Yaskawa INFORM job: aprem3TRJ4.JBI

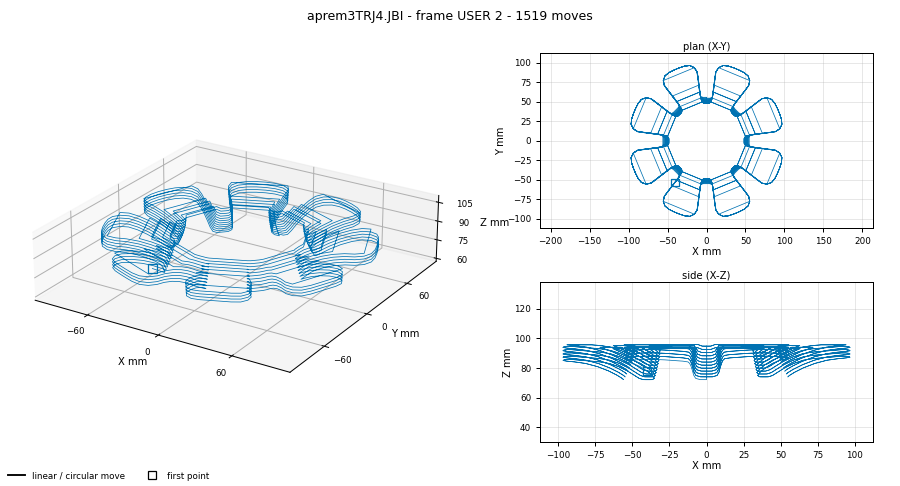
[picture p0: tool path of aprem3TRJ4.JBI in frame USER 2, 1519 of 1519 moves have a stored position in this frame; points joined in program order, loops and branches not executed]
/JOB
//NAME aprem3TRJ4
///FOLDERNAME DEMO
//POS
///NPOS 1519,0,1519,0,0,0
///USER 2
///TOOL 7
///POSTYPE USER
///RECTAN
///RCONF 1,0,0,0,0,0,0,0,0,0,0,0,0,0,0,0,0,0,0,0,0,0,0,0
C00000=-40.007,-53.324,78.036,177.7295,-3.1005,-14256.8795
C00001=-36.517,-48.718,75.143,178.8242,-1.7083,-14256.8537
C00002=-35.037,-45.351,73.015,-179.8825,17.3486,-14257.6887
C00003=-36.538,-42.505,72.166,160.0580,24.5520,-14260.6829
C00004=-38.303,-40.803,72.129,156.0408,22.3844,-14263.1899
C00005=-39.567,-39.567,72.154,156.8171,23.1818,-14265.0000
C00006=-40.803,-38.303,72.129,157.6162,23.9597,-14266.8101
C00007=-42.506,-36.538,72.166,155.4471,19.9396,-14269.3178
C00008=-45.352,-35.037,73.015,162.6519,-0.1179,-14272.3119
C00009=-48.718,-36.517,75.143,-178.2917,1.1758,-14273.1463
C00010=-53.324,-40.007,78.036,-176.8995,2.2705,-14273.1205
C00011=-59.196,-44.618,80.927,-176.4745,2.6327,-14272.9934
C00012=-65.578,-49.604,83.062,-176.2466,2.8111,-14272.8957
C00013=-71.524,-53.949,84.088,-176.0077,2.0393,-14272.9735
C00014=-77.795,-55.184,84.621,-177.1914,-0.2563,-14274.6500
C00015=-83.601,-53.037,85.050,-178.9039,-0.7847,-14277.6087
C00016=-87.741,-47.957,85.481,-179.9577,-0.0772,-14281.3401
C00017=-90.934,-41.602,85.762,-179.9958,-0.0092,-14285.4161
C00018=-93.717,-34.883,85.762,-179.9965,-0.0095,-14289.5839
C00019=-95.953,-28.131,85.481,-179.9754,-0.0845,-14293.6602
C00020=-96.617,-21.612,85.050,179.7797,-1.3299,-14297.3912
C00021=-94.030,-15.989,84.621,178.1943,-2.1678,-14300.3496
C00022=-88.723,-12.427,84.088,175.7377,-1.3847,-14302.0267
C00023=-81.446,-11.295,83.062,175.3629,-0.6685,-14302.1045
C00024=-73.408,-10.308,80.927,175.6494,-0.6331,-14302.0068
C00025=-65.995,-9.417,78.036,176.2047,-0.5882,-14301.8791
C00026=-60.270,-8.627,75.143,177.9610,-0.3768,-14301.8541
C00027=-56.844,-7.293,73.015,-167.4643,12.3773,-14302.6890
C00028=-55.892,-4.219,72.166,-176.1973,30.0956,-14305.6832
C00029=-55.936,-1.768,72.129,178.6826,31.1925,-14308.1896
C00030=-55.957,0.000,72.154,179.9991,31.1998,-14310.0000
C00031=-55.936,1.767,72.129,-178.6816,31.1926,-14311.8094
C00032=-55.892,4.220,72.166,176.1946,30.0948,-14314.3178
C00033=-56.844,7.293,73.015,167.4645,12.3766,-14317.3110
C00034=-60.270,8.627,75.143,-177.9610,-0.3768,-14318.1459
C00035=-65.995,9.417,78.036,-176.2047,-0.5882,-14318.1209
C00036=-73.408,10.308,80.927,-175.6494,-0.6331,-14317.9932
C00037=-81.446,11.295,83.062,-175.3629,-0.6685,-14317.8955
C00038=-88.723,12.427,84.088,-175.7377,-1.3847,-14317.9733
C00039=-94.030,15.989,84.621,-178.1943,-2.1678,-14319.6504
C00040=-96.617,21.612,85.050,-179.7797,-1.3299,-14322.6088
C00041=-95.953,28.131,85.481,179.9754,-0.0845,-14326.3398
C00042=-93.717,34.883,85.762,179.9965,-0.0095,-14330.4161
C00043=-90.934,41.602,85.762,179.9958,-0.0092,-14334.5839
C00044=-87.741,47.957,85.481,179.9577,-0.0772,-14338.6599
C00045=-83.601,53.037,85.050,178.9039,-0.7847,-14342.3913
C00046=-77.795,55.184,84.621,177.1914,-0.2563,-14345.3500
C00047=-71.524,53.949,84.088,176.0077,2.0393,-14347.0265
C00048=-65.578,49.604,83.062,176.2466,2.8111,-14347.1043
C00049=-59.196,44.618,80.927,176.4745,2.6327,-14347.0066
C00050=-53.324,40.007,78.036,176.8995,2.2705,-14346.8795
C00051=-48.718,36.517,75.143,178.2917,1.1758,-14346.8537
C00052=-45.351,35.037,73.015,-162.6514,-0.1175,-14347.6887
C00053=-42.505,36.538,72.166,-155.4480,19.9420,-14350.6829
C00054=-40.803,38.303,72.129,-157.6156,23.9592,-14353.1899
C00055=-39.567,39.567,72.154,-156.8182,23.1829,-14355.0000
C00056=-38.303,40.803,72.129,-156.0403,22.3838,-14356.8101
C00057=-36.538,42.506,72.166,-160.0604,24.5529,-14359.3178
C00058=-35.037,45.352,73.015,179.8821,17.3481,-14362.3119
C00059=-36.517,48.718,75.143,-178.8242,-1.7083,-14363.1463
C00060=-40.007,53.324,78.036,-177.7295,-3.1005,-14363.1205
C00061=-44.618,59.196,80.927,-177.3673,-3.5255,-14362.9934
C00062=-49.604,65.578,83.062,-177.1889,-3.7534,-14362.8957
C00063=-53.949,71.524,84.088,-177.9607,-3.9923,-14362.9735
C00064=-55.184,77.795,84.621,179.7437,-2.8086,-14364.6500
C00065=-53.037,83.601,85.050,179.2153,-1.0961,-14367.6087
C00066=-47.957,87.741,85.481,179.9228,-0.0423,-14371.3401
C00067=-41.602,90.934,85.762,179.9908,-0.0042,-14375.4161
C00068=-34.883,93.717,85.762,179.9905,-0.0035,-14379.5839
C00069=-28.131,95.953,85.481,179.9155,-0.0246,-14383.6602
C00070=-21.612,96.617,85.050,178.6701,0.2203,-14387.3912
C00071=-15.989,94.030,84.621,177.8322,1.8057,-14390.3496
C00072=-12.427,88.723,84.088,178.6153,4.2623,-14392.0267
C00073=-11.295,81.446,83.062,179.3315,4.6371,-14392.1045
C00074=-10.308,73.408,80.927,179.3669,4.3506,-14392.0068
C00075=-9.417,65.995,78.036,179.4118,3.7953,-14391.8791
C00076=-8.627,60.270,75.143,179.6232,2.0390,-14391.8541
C00077=-7.293,56.844,73.015,-167.6234,-12.5355,-14392.6890
C00078=-4.220,55.892,72.166,-149.9052,-3.8054,-14395.6822
C00079=-1.767,55.936,72.129,-148.8074,1.3184,-14398.1906
C00080=0.000,55.957,72.154,-148.8002,-0.0009,-14400.0000
C00081=0.000,54.840,74.049,-150.2606,-0.0009,-14400.0000
C00082=1.666,54.823,74.024,-150.2652,-1.1897,-14401.7406
C00083=4.048,54.790,74.062,-151.4249,3.8705,-14404.2255
C00084=7.088,55.804,74.943,-168.9167,11.6638,-14407.2387
C00085=8.393,59.388,77.145,179.6271,-2.1340,-14408.0440
C00086=9.180,65.335,80.122,179.4707,-3.5331,-14407.9981
C00087=10.089,72.980,83.074,179.4510,-3.8704,-14407.8709
C00088=11.094,81.206,85.240,179.4410,-3.9838,-14407.7793
C00089=12.226,88.613,86.276,178.8532,-3.5972,-14407.8555
C00090=15.808,94.009,86.813,178.1980,-1.5172,-14409.5452
C00091=21.475,96.642,87.246,178.9013,-0.1852,-14412.5282
C00092=28.048,95.980,87.679,179.9308,0.0202,-14416.2898
C00093=34.856,93.728,87.962,179.9923,0.0029,-14420.3994
C00094=41.629,90.922,87.962,179.9925,0.0034,-14424.6009
C00095=48.035,87.701,87.679,179.9368,0.0347,-14428.7101
C00096=53.151,83.521,87.246,179.3540,0.9079,-14432.4718
C00097=55.296,77.652,86.813,179.7985,2.3464,-14435.4547
C00098=54.014,71.304,86.276,-178.2646,3.3541,-14437.1446
C00099=49.577,65.266,85.240,-177.5752,3.2135,-14437.2208
C00100=44.470,58.738,83.074,-177.6486,3.1261,-14437.1290
C00101=39.708,52.690,80.122,-177.8738,2.8733,-14437.0022
C00102=36.059,47.928,77.145,-178.7542,1.7728,-14436.9563
C00103=34.447,44.472,74.943,179.5730,-15.8802,-14437.7605
C00104=35.880,41.605,74.062,-161.3614,-23.4111,-14440.7744
C00105=37.588,39.944,74.024,-157.2868,-21.2665,-14443.2595
C00106=38.778,38.778,74.049,-158.0022,-21.9968,-14445.0000
C00107=39.943,37.588,74.024,-158.7340,-22.7138,-14446.7398
C00108=41.605,35.880,74.062,-156.5881,-18.6363,-14449.2256
C00109=44.472,34.447,74.943,-164.1205,0.4274,-14452.2395
C00110=47.928,36.059,77.145,178.2272,-1.2458,-14453.0437
C00111=52.690,39.708,80.122,177.1267,-2.1262,-14452.9978
C00112=58.738,44.470,83.074,176.8739,-2.3514,-14452.8710
C00113=65.266,49.577,85.240,176.7865,-2.4248,-14452.7792
C00114=71.304,54.014,86.276,176.6459,-1.7354,-14452.8554
C00115=77.652,55.296,86.813,177.6536,0.2015,-14454.5453
C00116=83.521,53.151,87.246,179.0921,0.6460,-14457.5282
C00117=87.701,48.035,87.679,179.9653,0.0632,-14461.2899
C00118=90.922,41.629,87.962,179.9966,0.0075,-14465.3991
C00119=93.728,34.856,87.962,179.9971,0.0077,-14469.6006
C00120=95.980,28.048,87.679,179.9798,0.0692,-14473.7102
C00121=96.642,21.475,87.246,-179.8148,1.0987,-14477.4718
C00122=94.009,15.808,86.813,-178.4828,1.8020,-14480.4548
C00123=88.613,12.226,86.276,-176.4028,1.1468,-14482.1445
C00124=81.206,11.094,85.240,-176.0162,0.5590,-14482.2207
C00125=72.980,10.089,83.074,-176.1296,0.5490,-14482.1291
C00126=65.335,9.180,80.122,-176.4669,0.5293,-14482.0019
C00127=59.388,8.393,77.145,-177.8660,0.3729,-14481.9560
C00128=55.804,7.088,74.943,168.3362,-11.0833,-14482.7613
C00129=54.790,4.048,74.062,176.1295,-28.5751,-14485.7745
C00130=54.823,1.666,74.024,-178.8103,-29.7348,-14488.2594
C00131=54.840,0.000,74.049,-179.9991,-29.7394,-14490.0000
C00132=54.823,-1.665,74.024,178.8094,-29.7348,-14491.7396
C00133=54.790,-4.048,74.062,-176.1270,-28.5741,-14494.2255
C00134=55.804,-7.088,74.943,-168.3364,-11.0826,-14497.2387
C00135=59.388,-8.393,77.145,177.8660,0.3729,-14498.0440
C00136=65.335,-9.180,80.122,176.4669,0.5293,-14497.9981
C00137=72.980,-10.089,83.074,176.1296,0.5490,-14497.8709
C00138=81.206,-11.094,85.240,176.0162,0.5590,-14497.7793
C00139=88.613,-12.226,86.276,176.4028,1.1468,-14497.8555
C00140=94.009,-15.808,86.813,178.4828,1.8020,-14499.5452
C00141=96.642,-21.475,87.246,179.8148,1.0987,-14502.5282
C00142=95.980,-28.048,87.679,-179.9798,0.0692,-14506.2898
C00143=93.728,-34.856,87.962,-179.9971,0.0077,-14510.3994
C00144=90.922,-41.629,87.962,-179.9966,0.0075,-14514.6009
C00145=87.701,-48.035,87.679,-179.9653,0.0632,-14518.7101
C00146=83.521,-53.151,87.246,-179.0921,0.6460,-14522.4718
C00147=77.652,-55.296,86.813,-177.6536,0.2015,-14525.4547
C00148=71.304,-54.014,86.276,-176.6459,-1.7354,-14527.1446
C00149=65.266,-49.577,85.240,-176.7865,-2.4248,-14527.2208
C00150=58.738,-44.470,83.074,-176.8739,-2.3514,-14527.1290
C00151=52.690,-39.708,80.122,-177.1267,-2.1262,-14527.0022
C00152=47.928,-36.059,77.145,-178.2272,-1.2458,-14526.9563
C00153=44.472,-34.447,74.943,164.1198,0.4270,-14527.7605
C00154=41.605,-35.880,74.062,156.5889,-18.6386,-14530.7744
C00155=39.944,-37.588,74.024,158.7335,-22.7132,-14533.2595
C00156=38.778,-38.778,74.049,158.0032,-21.9978,-14535.0000
C00157=37.588,-39.943,74.024,157.2862,-21.2660,-14536.7398
C00158=35.880,-41.605,74.062,161.3637,-23.4119,-14539.2256
C00159=34.447,-44.472,74.943,-179.5726,-15.8795,-14542.2395
C00160=36.059,-47.928,77.145,178.7542,1.7728,-14543.0437
C00161=39.708,-52.690,80.122,177.8738,2.8733,-14542.9978
C00162=44.470,-58.738,83.074,177.6486,3.1261,-14542.8710
C00163=49.577,-65.266,85.240,177.5752,3.2135,-14542.7792
C00164=54.014,-71.304,86.276,178.2646,3.3541,-14542.8554
C00165=55.296,-77.652,86.813,-179.7985,2.3464,-14544.5453
C00166=53.151,-83.521,87.246,-179.3540,0.9079,-14547.5282
C00167=48.035,-87.701,87.679,-179.9368,0.0347,-14551.2899
C00168=41.629,-90.922,87.962,-179.9925,0.0034,-14555.3991
C00169=34.856,-93.728,87.962,-179.9923,0.0029,-14559.6006
C00170=28.048,-95.980,87.679,-179.9308,0.0202,-14563.7102
C00171=21.475,-96.642,87.246,-178.9013,-0.1852,-14567.4718
C00172=15.808,-94.009,86.813,-178.1980,-1.5172,-14570.4548
C00173=12.226,-88.613,86.276,-178.8532,-3.5972,-14572.1445
C00174=11.094,-81.206,85.240,-179.4410,-3.9838,-14572.2207
C00175=10.089,-72.980,83.074,-179.4510,-3.8704,-14572.1291
C00176=9.180,-65.335,80.122,-179.4707,-3.5331,-14572.0019
C00177=8.393,-59.388,77.145,-179.6271,-2.1340,-14571.9560
C00178=7.088,-55.804,74.943,168.9167,11.6638,-14572.7613
C00179=4.048,-54.790,74.062,151.4249,3.8705,-14575.7745
C00180=1.666,-54.823,74.024,150.2652,-1.1897,-14578.2594
C00181=0.000,-54.840,74.049,150.2606,-0.0009,-14580.0000
C00182=0.000,-54.840,74.049,150.2606,-0.0009,-14580.0000
C00183=-1.665,-54.823,74.024,150.2652,1.1906,-14581.7396
C00184=-4.048,-54.790,74.062,151.4259,-3.8730,-14584.2255
C00185=-7.088,-55.804,74.943,168.9174,-11.6636,-14587.2387
C00186=-8.393,-59.388,77.145,-179.6271,2.1340,-14588.0440
C00187=-9.180,-65.335,80.122,-179.4707,3.5331,-14587.9981
C00188=-10.089,-72.980,83.074,-179.4510,3.8704,-14587.8709
C00189=-11.094,-81.206,85.240,-179.4410,3.9838,-14587.7793
C00190=-12.226,-88.613,86.276,-178.8532,3.5972,-14587.8555
C00191=-15.808,-94.009,86.813,-178.1980,1.5172,-14589.5452
C00192=-21.475,-96.642,87.246,-178.9013,0.1852,-14592.5282
C00193=-28.048,-95.980,87.679,-179.9308,-0.0202,-14596.2898
C00194=-34.856,-93.728,87.962,-179.9923,-0.0029,-14600.3994
C00195=-41.629,-90.922,87.962,-179.9925,-0.0034,-14604.6009
C00196=-48.035,-87.701,87.679,-179.9368,-0.0347,-14608.7101
C00197=-53.151,-83.521,87.246,-179.3540,-0.9079,-14612.4718
C00198=-55.296,-77.652,86.813,-179.7985,-2.3464,-14615.4547
C00199=-54.014,-71.304,86.276,178.2646,-3.3541,-14617.1446
C00200=-49.577,-65.266,85.240,177.5752,-3.2135,-14617.2208
C00201=-44.470,-58.738,83.074,177.6486,-3.1261,-14617.1290
C00202=-39.708,-52.690,80.122,177.8738,-2.8733,-14617.0022
C00203=-36.059,-47.928,77.145,178.7542,-1.7728,-14616.9563
C00204=-34.447,-44.472,74.943,-179.5730,15.8802,-14617.7605
C00205=-35.880,-41.605,74.062,161.3614,23.4111,-14620.7744
C00206=-37.588,-39.944,74.024,157.2868,21.2665,-14623.2595
C00207=-38.778,-38.778,74.049,158.0022,21.9968,-14625.0000
C00208=-39.943,-37.588,74.024,158.7340,22.7138,-14626.7398
C00209=-41.605,-35.880,74.062,156.5881,18.6363,-14629.2256
C00210=-44.472,-34.447,74.943,164.1205,-0.4274,-14632.2395
C00211=-47.928,-36.059,77.145,-178.2272,1.2458,-14633.0437
C00212=-52.690,-39.708,80.122,-177.1267,2.1262,-14632.9978
C00213=-58.738,-44.470,83.074,-176.8739,2.3514,-14632.8710
C00214=-65.266,-49.577,85.240,-176.7865,2.4248,-14632.7792
C00215=-71.304,-54.014,86.276,-176.6459,1.7354,-14632.8554
C00216=-77.652,-55.296,86.813,-177.6536,-0.2015,-14634.5453
C00217=-83.521,-53.151,87.246,-179.0921,-0.6460,-14637.5282
C00218=-87.701,-48.035,87.679,-179.9653,-0.0632,-14641.2899
C00219=-90.922,-41.629,87.962,-179.9966,-0.0075,-14645.3991
C00220=-93.728,-34.856,87.962,-179.9971,-0.0077,-14649.6006
C00221=-95.980,-28.048,87.679,-179.9798,-0.0692,-14653.7102
C00222=-96.642,-21.475,87.246,179.8148,-1.0987,-14657.4718
C00223=-94.009,-15.808,86.813,178.4828,-1.8020,-14660.4548
C00224=-88.613,-12.226,86.276,176.4028,-1.1468,-14662.1445
C00225=-81.206,-11.094,85.240,176.0162,-0.5590,-14662.2207
C00226=-72.980,-10.089,83.074,176.1296,-0.5490,-14662.1291
C00227=-65.335,-9.180,80.122,176.4669,-0.5293,-14662.0019
C00228=-59.388,-8.393,77.145,177.8660,-0.3729,-14661.9560
C00229=-55.804,-7.088,74.943,-168.3362,11.0833,-14662.7613
C00230=-54.790,-4.048,74.062,-176.1295,28.5751,-14665.7745
C00231=-54.823,-1.666,74.024,178.8103,29.7348,-14668.2594
C00232=-54.840,0.000,74.049,179.9991,29.7394,-14670.0000
C00233=-54.823,1.665,74.024,-178.8094,29.7348,-14671.7396
C00234=-54.790,4.048,74.062,176.1270,28.5741,-14674.2255
C00235=-55.804,7.088,74.943,168.3364,11.0826,-14677.2387
C00236=-59.388,8.393,77.145,-177.8660,-0.3729,-14678.0440
C00237=-65.335,9.180,80.122,-176.4669,-0.5293,-14677.9981
C00238=-72.980,10.089,83.074,-176.1296,-0.5490,-14677.8709
C00239=-81.206,11.094,85.240,-176.0162,-0.5590,-14677.7793
C00240=-88.613,12.226,86.276,-176.4028,-1.1468,-14677.8555
C00241=-94.009,15.808,86.813,-178.4828,-1.8020,-14679.5452
C00242=-96.642,21.475,87.246,-179.8148,-1.0987,-14682.5282
C00243=-95.980,28.048,87.679,179.9798,-0.0692,-14686.2898
C00244=-93.728,34.856,87.962,179.9971,-0.0077,-14690.3994
C00245=-90.922,41.629,87.962,179.9966,-0.0075,-14694.6009
C00246=-87.701,48.035,87.679,179.9653,-0.0632,-14698.7101
C00247=-83.521,53.151,87.246,179.0921,-0.6460,-14702.4718
C00248=-77.652,55.296,86.813,177.6536,-0.2015,-14705.4547
C00249=-71.304,54.014,86.276,176.6459,1.7354,-14707.1446
C00250=-65.266,49.577,85.240,176.7865,2.4248,-14707.2208
C00251=-58.738,44.470,83.074,176.8739,2.3514,-14707.1290
C00252=-52.690,39.708,80.122,177.1267,2.1262,-14707.0022
C00253=-47.928,36.059,77.145,178.2272,1.2458,-14706.9563
C00254=-44.472,34.447,74.943,-164.1198,-0.4270,-14707.7605
C00255=-41.605,35.880,74.062,-156.5889,18.6386,-14710.7744
C00256=-39.944,37.588,74.024,-158.7335,22.7132,-14713.2595
C00257=-38.778,38.778,74.049,-158.0032,21.9978,-14715.0000
C00258=-37.588,39.943,74.024,-157.2862,21.2660,-14716.7398
C00259=-35.880,41.605,74.062,-161.3637,23.4119,-14719.2256
C00260=-34.447,44.472,74.943,179.5726,15.8795,-14722.2395
C00261=-36.059,47.928,77.145,-178.7542,-1.7728,-14723.0437
C00262=-39.708,52.690,80.122,-177.8738,-2.8733,-14722.9978
C00263=-44.470,58.738,83.074,-177.6486,-3.1261,-14722.8710
C00264=-49.577,65.266,85.240,-177.5752,-3.2135,-14722.7792
C00265=-54.014,71.304,86.276,-178.2646,-3.3541,-14722.8554
C00266=-55.296,77.652,86.813,179.7985,-2.3464,-14724.5453
C00267=-53.151,83.521,87.246,179.3540,-0.9079,-14727.5282
C00268=-48.035,87.701,87.679,179.9368,-0.0347,-14731.2899
C00269=-41.629,90.922,87.962,179.9925,-0.0034,-14735.3991
C00270=-34.856,93.728,87.962,179.9923,-0.0029,-14739.6006
C00271=-28.048,95.980,87.679,179.9308,-0.0202,-14743.7102
C00272=-21.475,96.642,87.246,178.9013,0.1852,-14747.4718
C00273=-15.808,94.009,86.813,178.1980,1.5172,-14750.4548
C00274=-12.226,88.613,86.276,178.8532,3.5972,-14752.1445
C00275=-11.094,81.206,85.240,179.4410,3.9838,-14752.2207
C00276=-10.089,72.980,83.074,179.4510,3.8704,-14752.1291
C00277=-9.180,65.335,80.122,179.4707,3.5331,-14752.0019
C00278=-8.393,59.388,77.145,179.6271,2.1340,-14751.9560
C00279=-7.088,55.804,74.943,-168.9174,-11.6636,-14752.7613
C00280=-4.048,54.790,74.062,-151.4259,-3.8730,-14755.7745
C00281=-1.665,54.823,74.024,-150.2652,1.1906,-14758.2604
C00282=0.000,54.840,74.049,-150.2606,-0.0009,-14760.0000
C00283=0.000,53.776,75.975,-151.9017,-0.0008,-14760.0000
C00284=1.568,53.762,75.948,-151.9034,-1.0593,-14761.6706
C00285=3.884,53.739,75.988,-153.1148,3.8750,-14764.1339
C00286=6.894,54.818,76.900,-170.1649,10.7294,-14767.1680
C00287=8.175,58.565,79.173,179.6434,-2.1517,-14767.9465
C00288=8.965,64.737,82.228,179.5331,-3.2135,-14767.8844
C00289=9.898,72.606,85.234,179.5371,-3.3364,-14767.7630
C00290=10.924,81.005,87.424,179.5509,-3.2738,-14767.6803
C00291=12.061,88.524,88.468,179.0976,-2.8742,-14767.7585
C00292=15.662,93.991,89.008,178.5900,-1.1973,-14769.4604
C00293=21.365,96.662,89.443,179.1515,-0.1450,-14772.4636
C00294=27.983,96.002,89.878,179.9474,0.0153,-14776.2505
C00295=34.834,93.736,90.162,179.9942,0.0022,-14780.3860
C00296=41.650,90.913,90.162,179.9944,0.0026,-14784.6140
C00297=48.097,87.670,89.878,179.9520,0.0264,-14788.7498
C00298=53.243,83.458,89.443,179.5025,0.7025,-14792.5363
C00299=55.387,77.537,89.008,179.8495,1.8433,-14795.5394
C00300=54.067,71.124,88.468,-178.6043,2.6703,-14797.2413
C00301=49.554,65.004,87.424,-178.0010,2.6331,-14797.3191
C00302=44.341,58.339,85.234,-177.9664,2.6872,-14797.2369
C00303=39.437,52.115,82.228,-178.0562,2.6030,-14797.1159
C00304=35.631,47.192,79.173,-178.7302,1.7738,-14797.0536
C00305=33.888,43.637,76.900,179.3468,-14.3899,-14797.8325
C00306=35.253,40.746,75.988,-162.7447,-22.1169,-14800.8660
C00307=36.906,39.124,75.948,-158.6653,-20.0234,-14803.3290
C00308=38.025,38.025,75.975,-159.3164,-20.6826,-14805.0000
C00309=39.124,36.906,75.948,-159.9771,-21.3352,-14806.6710
C00310=40.746,35.253,75.988,-157.8823,-17.2529,-14809.1340
C00311=43.637,33.888,76.901,-165.6107,0.6536,-14812.1675
C00312=47.192,35.631,79.173,178.2262,-1.2698,-14812.9464
C00313=52.115,39.437,82.228,177.3970,-1.9438,-14812.8841
C00314=58.339,44.341,85.234,177.3128,-2.0336,-14812.7631
C00315=65.004,49.554,87.424,177.3669,-1.9990,-14812.6809
C00316=71.124,54.067,88.468,177.3297,-1.3957,-14812.7587
C00317=77.537,55.387,89.008,178.1567,0.1505,-14814.4606
C00318=83.458,53.243,89.443,179.2975,0.4975,-14817.4637
C00319=87.670,48.097,89.878,179.9736,0.0480,-14821.2502
C00320=90.913,41.650,90.162,179.9974,0.0056,-14825.3860
C00321=93.736,34.834,90.162,179.9978,0.0058,-14829.6140
C00322=96.002,27.983,89.878,179.9847,0.0526,-14833.7495
C00323=96.662,21.365,89.443,-179.8550,0.8485,-14837.5364
C00324=93.991,15.662,89.008,-178.8027,1.4100,-14840.5396
C00325=88.524,12.061,88.468,-177.1258,0.9024,-14842.2415
C00326=81.005,10.924,87.424,-176.7262,0.4491,-14842.3197
C00327=72.606,9.898,85.234,-176.6636,0.4629,-14842.2370
C00328=64.737,8.965,82.228,-176.7865,0.4669,-14842.1156
C00329=58.565,8.175,79.173,-177.8483,0.3566,-14842.0535
C00330=54.818,6.894,76.900,169.2706,-9.8351,-14842.8320
C00331=53.739,3.884,75.988,176.1250,-26.8852,-14845.8661
C00332=53.762,1.568,75.948,-178.9407,-28.0966,-14848.3294
C00333=53.776,0.000,75.975,-179.9992,-28.0983,-14850.0000
C00334=53.762,-1.568,75.948,178.9399,-28.0967,-14851.6706
C00335=53.739,-3.885,75.988,-176.1225,-26.8842,-14854.1349
C00336=54.819,-6.894,76.901,-169.2709,-9.8343,-14857.1678
C00337=58.565,-8.175,79.173,177.8483,0.3566,-14857.9465
C00338=64.737,-8.965,82.228,176.7865,0.4669,-14857.8844
C00339=72.606,-9.898,85.234,176.6636,0.4629,-14857.7630
C00340=81.005,-10.924,87.424,176.7262,0.4491,-14857.6803
C00341=88.524,-12.061,88.468,177.1258,0.9024,-14857.7585
C00342=93.991,-15.662,89.008,178.8027,1.4100,-14859.4604
C00343=96.662,-21.365,89.443,179.8550,0.8485,-14862.4636
C00344=96.002,-27.983,89.878,-179.9847,0.0526,-14866.2505
C00345=93.736,-34.834,90.162,-179.9978,0.0058,-14870.3860
C00346=90.913,-41.650,90.162,-179.9974,0.0056,-14874.6140
C00347=87.670,-48.097,89.878,-179.9736,0.0480,-14878.7498
C00348=83.458,-53.243,89.443,-179.2975,0.4975,-14882.5363
C00349=77.537,-55.387,89.008,-178.1567,0.1505,-14885.5394
C00350=71.124,-54.067,88.468,-177.3297,-1.3957,-14887.2413
C00351=65.004,-49.554,87.424,-177.3669,-1.9990,-14887.3191
C00352=58.339,-44.341,85.234,-177.3128,-2.0336,-14887.2369
C00353=52.115,-39.437,82.228,-177.3970,-1.9438,-14887.1159
C00354=47.192,-35.631,79.173,-178.2262,-1.2698,-14887.0536
C00355=43.637,-33.888,76.900,165.6101,0.6532,-14887.8325
C00356=40.746,-35.253,75.988,157.8831,-17.2553,-14890.8660
C00357=39.124,-36.906,75.948,159.9766,-21.3347,-14893.3290
C00358=38.025,-38.025,75.975,159.3174,-20.6836,-14895.0000
C00359=36.906,-39.124,75.948,158.6648,-20.0229,-14896.6710
C00360=35.253,-40.746,75.988,162.7471,-22.1177,-14899.1340
C00361=33.888,-43.637,76.901,-179.3464,-14.3893,-14902.1675
C00362=35.631,-47.192,79.173,178.7302,1.7738,-14902.9464
C00363=39.437,-52.115,82.228,178.0562,2.6030,-14902.8841
C00364=44.341,-58.339,85.234,177.9664,2.6872,-14902.7631
C00365=49.554,-65.004,87.424,178.0010,2.6331,-14902.6809
C00366=54.067,-71.124,88.468,178.6043,2.6703,-14902.7587
C00367=55.387,-77.537,89.008,-179.8495,1.8433,-14904.4606
C00368=53.243,-83.458,89.443,-179.5025,0.7025,-14907.4637
C00369=48.097,-87.670,89.878,-179.9520,0.0264,-14911.2502
C00370=41.650,-90.913,90.162,-179.9944,0.0026,-14915.3860
C00371=34.834,-93.736,90.162,-179.9942,0.0022,-14919.6140
C00372=27.983,-96.002,89.878,-179.9474,0.0153,-14923.7495
C00373=21.365,-96.662,89.443,-179.1515,-0.1450,-14927.5364
C00374=15.662,-93.991,89.008,-178.5900,-1.1973,-14930.5396
C00375=12.061,-88.524,88.468,-179.0976,-2.8742,-14932.2415
C00376=10.924,-81.005,87.424,-179.5509,-3.2738,-14932.3197
C00377=9.898,-72.606,85.234,-179.5371,-3.3364,-14932.2370
C00378=8.965,-64.737,82.228,-179.5331,-3.2135,-14932.1156
C00379=8.175,-58.565,79.173,-179.6434,-2.1517,-14932.0535
C00380=6.894,-54.818,76.900,170.1649,10.7294,-14932.8320
C00381=3.884,-53.739,75.988,153.1148,3.8750,-14935.8661
C00382=1.568,-53.762,75.948,151.9034,-1.0593,-14938.3294
C00383=0.000,-53.776,75.975,151.9017,-0.0008,-14940.0000
C00384=0.000,-53.776,75.975,151.9017,-0.0008,-14940.0000
C00385=-1.568,-53.762,75.948,151.9033,1.0601,-14941.6706
C00386=-3.885,-53.739,75.988,153.1158,-3.8775,-14944.1349
C00387=-6.894,-54.819,76.901,170.1657,-10.7291,-14947.1678
C00388=-8.175,-58.565,79.173,-179.6434,2.1517,-14947.9465
C00389=-8.965,-64.737,82.228,-179.5331,3.2135,-14947.8844
C00390=-9.898,-72.606,85.234,-179.5371,3.3364,-14947.7630
C00391=-10.924,-81.005,87.424,-179.5509,3.2738,-14947.6803
C00392=-12.061,-88.524,88.468,-179.0976,2.8742,-14947.7585
C00393=-15.662,-93.991,89.008,-178.5900,1.1973,-14949.4604
C00394=-21.365,-96.662,89.443,-179.1515,0.1450,-14952.4636
C00395=-27.983,-96.002,89.878,-179.9474,-0.0153,-14956.2505
C00396=-34.834,-93.736,90.162,-179.9942,-0.0022,-14960.3860
C00397=-41.650,-90.913,90.162,-179.9944,-0.0026,-14964.6140
C00398=-48.097,-87.670,89.878,-179.9520,-0.0264,-14968.7498
C00399=-53.243,-83.458,89.443,-179.5025,-0.7025,-14972.5363
C00400=-55.387,-77.537,89.008,-179.8495,-1.8433,-14975.5394
C00401=-54.067,-71.124,88.468,178.6043,-2.6703,-14977.2413
C00402=-49.554,-65.004,87.424,178.0010,-2.6331,-14977.3191
C00403=-44.341,-58.339,85.234,177.9664,-2.6872,-14977.2369
C00404=-39.437,-52.115,82.228,178.0562,-2.6030,-14977.1159
C00405=-35.631,-47.192,79.173,178.7302,-1.7738,-14977.0536
C00406=-33.888,-43.637,76.900,-179.3468,14.3899,-14977.8325
C00407=-35.253,-40.746,75.988,162.7447,22.1169,-14980.8660
C00408=-36.906,-39.124,75.948,158.6653,20.0234,-14983.3290
C00409=-38.025,-38.025,75.975,159.3164,20.6826,-14985.0000
C00410=-39.124,-36.906,75.948,159.9771,21.3352,-14986.6710
C00411=-40.746,-35.253,75.988,157.8823,17.2529,-14989.1340
C00412=-43.637,-33.888,76.901,165.6107,-0.6536,-14992.1675
C00413=-47.192,-35.631,79.173,-178.2262,1.2698,-14992.9464
C00414=-52.115,-39.437,82.228,-177.3970,1.9438,-14992.8841
C00415=-58.339,-44.341,85.234,-177.3128,2.0336,-14992.7631
C00416=-65.004,-49.554,87.424,-177.3669,1.9990,-14992.6809
C00417=-71.124,-54.067,88.468,-177.3297,1.3957,-14992.7587
C00418=-77.537,-55.387,89.008,-178.1567,-0.1505,-14994.4606
C00419=-83.458,-53.243,89.443,-179.2975,-0.4975,-14997.4637
C00420=-87.670,-48.097,89.878,-179.9736,-0.0480,-15001.2502
C00421=-90.913,-41.650,90.162,-179.9974,-0.0056,-15005.3860
C00422=-93.736,-34.834,90.162,-179.9978,-0.0058,-15009.6140
C00423=-96.002,-27.983,89.878,-179.9847,-0.0526,-15013.7495
C00424=-96.662,-21.365,89.443,179.8550,-0.8485,-15017.5364
C00425=-93.991,-15.662,89.008,178.8027,-1.4100,-15020.5396
C00426=-88.524,-12.061,88.468,177.1258,-0.9024,-15022.2415
C00427=-81.005,-10.924,87.424,176.7262,-0.4491,-15022.3197
C00428=-72.606,-9.898,85.234,176.6636,-0.4629,-15022.2370
C00429=-64.737,-8.965,82.228,176.7865,-0.4669,-15022.1156
C00430=-58.565,-8.175,79.173,177.8483,-0.3566,-15022.0535
C00431=-54.818,-6.894,76.900,-169.2706,9.8351,-15022.8320
C00432=-53.739,-3.884,75.988,-176.1250,26.8852,-15025.8661
C00433=-53.762,-1.568,75.948,178.9407,28.0966,-15028.3294
C00434=-53.776,0.000,75.975,179.9992,28.0983,-15030.0000
C00435=-53.762,1.568,75.948,-178.9399,28.0967,-15031.6706
C00436=-53.739,3.885,75.988,176.1225,26.8842,-15034.1349
C00437=-54.819,6.894,76.901,169.2709,9.8343,-15037.1678
C00438=-58.565,8.175,79.173,-177.8483,-0.3566,-15037.9465
C00439=-64.737,8.965,82.228,-176.7865,-0.4669,-15037.8844
C00440=-72.606,9.898,85.234,-176.6636,-0.4629,-15037.7630
C00441=-81.005,10.924,87.424,-176.7262,-0.4491,-15037.6803
C00442=-88.524,12.061,88.468,-177.1258,-0.9024,-15037.7585
C00443=-93.991,15.662,89.008,-178.8027,-1.4100,-15039.4604
C00444=-96.662,21.365,89.443,-179.8550,-0.8485,-15042.4636
C00445=-96.002,27.983,89.878,179.9847,-0.0526,-15046.2505
C00446=-93.736,34.834,90.162,179.9978,-0.0058,-15050.3860
C00447=-90.913,41.650,90.162,179.9974,-0.0056,-15054.6140
C00448=-87.670,48.097,89.878,179.9736,-0.0480,-15058.7498
C00449=-83.458,53.243,89.443,179.2975,-0.4975,-15062.5363
C00450=-77.537,55.387,89.008,178.1567,-0.1505,-15065.5394
C00451=-71.124,54.067,88.468,177.3297,1.3957,-15067.2413
C00452=-65.004,49.554,87.424,177.3669,1.9990,-15067.3191
C00453=-58.339,44.341,85.234,177.3128,2.0336,-15067.2369
C00454=-52.115,39.437,82.228,177.3970,1.9438,-15067.1159
C00455=-47.192,35.631,79.173,178.2262,1.2698,-15067.0536
C00456=-43.637,33.888,76.900,-165.6101,-0.6532,-15067.8325
C00457=-40.746,35.253,75.988,-157.8831,17.2553,-15070.8660
C00458=-39.124,36.906,75.948,-159.9766,21.3347,-15073.3290
C00459=-38.025,38.025,75.975,-159.3174,20.6836,-15075.0000
C00460=-36.906,39.124,75.948,-158.6648,20.0229,-15076.6710
C00461=-35.253,40.746,75.988,-162.7471,22.1177,-15079.1340
C00462=-33.888,43.637,76.901,179.3464,14.3893,-15082.1675
C00463=-35.631,47.192,79.173,-178.7302,-1.7738,-15082.9464
C00464=-39.437,52.115,82.228,-178.0562,-2.6030,-15082.8841
C00465=-44.341,58.339,85.234,-177.9664,-2.6872,-15082.7631
C00466=-49.554,65.004,87.424,-178.0010,-2.6331,-15082.6809
C00467=-54.067,71.124,88.468,-178.6043,-2.6703,-15082.7587
C00468=-55.387,77.537,89.008,179.8495,-1.8433,-15084.4606
C00469=-53.243,83.458,89.443,179.5025,-0.7025,-15087.4637
C00470=-48.097,87.670,89.878,179.9520,-0.0264,-15091.2502
C00471=-41.650,90.913,90.162,179.9944,-0.0026,-15095.3860
C00472=-34.834,93.736,90.162,179.9942,-0.0022,-15099.6140
C00473=-27.983,96.002,89.878,179.9474,-0.0153,-15103.7495
C00474=-21.365,96.662,89.443,179.1515,0.1450,-15107.5364
C00475=-15.662,93.991,89.008,178.5900,1.1973,-15110.5396
C00476=-12.061,88.524,88.468,179.0976,2.8742,-15112.2415
C00477=-10.924,81.005,87.424,179.5509,3.2738,-15112.3197
C00478=-9.898,72.606,85.234,179.5371,3.3364,-15112.2370
C00479=-8.965,64.737,82.228,179.5331,3.2135,-15112.1156
C00480=-8.175,58.565,79.173,179.6434,2.1517,-15112.0535
C00481=-6.894,54.819,76.901,-170.1657,-10.7291,-15112.8322
C00482=-3.885,53.739,75.988,-153.1158,-3.8775,-15115.8651
C00483=-1.568,53.762,75.948,-151.9033,1.0601,-15118.3294
C00484=0.000,53.776,75.975,-151.9017,-0.0008,-15120.0000
C00485=0.000,52.771,77.932,-153.7423,-0.0007,-15120.0000
C00486=1.476,52.759,77.904,-153.7405,-0.9277,-15121.6025
C00487=3.730,52.747,77.945,-154.9876,3.8100,-15124.0449
C00488=6.711,53.894,78.888,-171.3670,9.7384,-15127.0981
C00489=7.974,57.808,81.229,179.6695,-2.0942,-15127.8538
C00490=8.774,64.206,84.354,179.5987,-2.8379,-15127.7815
C00491=9.737,72.291,87.405,179.6254,-2.7503,-15127.6711
C00492=10.790,80.844,89.614,179.6620,-2.5088,-15127.6022
C00493=11.935,88.455,90.663,179.3495,-2.0963,-15127.6844
C00494=15.553,93.978,91.206,179.0073,-0.8482,-15129.3971
C00495=21.285,96.677,91.642,179.4198,-0.1001,-15132.4165
C00496=27.936,96.017,92.077,179.9653,0.0101,-15136.2223
C00497=34.820,93.742,92.362,179.9963,0.0014,-15140.3773
C00498=41.664,90.907,92.362,179.9964,0.0017,-15144.6227
C00499=48.140,87.648,92.077,179.9683,0.0174,-15148.7775
C00500=53.310,83.412,91.642,179.6605,0.4810,-15152.5833
C00501=55.455,77.451,91.206,179.8978,1.3016,-15155.6027
C00502=54.108,70.986,90.663,-178.9772,1.9422,-15157.3159
C00503=49.536,64.795,89.614,-178.4643,2.0133,-15157.3980
C00504=44.233,58.003,87.405,-178.3191,2.2100,-15157.3291
C00505=39.197,51.604,84.354,-178.2760,2.2909,-15157.2193
C00506=35.238,46.514,81.229,-178.7524,1.7146,-15157.1468
C00507=33.363,42.854,78.888,179.1980,-12.8827,-15157.9017
C00508=34.660,39.935,77.945,-164.2077,-20.6567,-15160.9551
C00509=36.262,38.350,77.904,-160.1858,-18.6445,-15163.3970
C00510=37.314,37.314,77.932,-160.7695,-19.2296,-15165.0000
C00511=38.350,36.262,77.904,-161.3560,-19.8147,-15166.6030
C00512=39.935,34.660,77.945,-159.3426,-15.7900,-15169.0449
C00513=42.854,33.363,78.888,-167.1181,0.8024,-15172.0983
C00514=46.514,35.238,81.229,178.2854,-1.2476,-15172.8532
C00515=51.604,39.197,84.354,177.7091,-1.7240,-15172.7807
C00516=58.003,44.233,87.405,177.7900,-1.6809,-15172.6709
C00517=64.795,49.536,89.614,177.9867,-1.5357,-15172.6020
C00518=70.986,54.108,90.663,178.0578,-1.0228,-15172.6841
C00519=77.451,55.455,91.206,178.6984,0.1022,-15174.3973
C00520=83.412,53.310,91.642,179.5190,0.3395,-15177.4167
C00521=87.648,48.140,92.077,179.9826,0.0317,-15181.2225
C00522=90.907,41.664,92.362,179.9983,0.0036,-15185.3773
C00523=93.742,34.820,92.362,179.9986,0.0037,-15189.6227
C00524=96.017,27.936,92.077,179.9899,0.0347,-15193.7777
C00525=96.677,21.285,91.642,-179.8999,0.5802,-15197.5835
C00526=93.978,15.553,91.206,-179.1518,0.9927,-15200.6029
C00527=88.455,11.935,90.663,-177.9037,0.6505,-15202.3156
C00528=80.844,10.790,89.614,-177.4912,0.3380,-15202.3978
C00529=72.291,9.737,87.405,-177.2497,0.3746,-15202.3289
C00530=64.206,8.774,84.354,-177.1621,0.4013,-15202.2185
C00531=57.808,7.974,81.229,-177.9058,0.3305,-15202.1462
C00532=53.894,6.711,78.888,170.2616,-8.6330,-15202.9019
C00533=52.747,3.730,77.945,176.1900,-25.0124,-15205.9551
C00534=52.759,1.476,77.904,-179.0723,-26.2595,-15208.3975
C00535=52.771,0.000,77.932,-179.9993,-26.2577,-15210.0000
C00536=52.759,-1.476,77.904,179.0716,-26.2595,-15211.6025
C00537=52.747,-3.730,77.945,-176.1877,-25.0114,-15214.0449
C00538=53.894,-6.711,78.888,-170.2619,-8.6323,-15217.0981
C00539=57.808,-7.974,81.229,177.9058,0.3305,-15217.8538
C00540=64.206,-8.774,84.354,177.1621,0.4013,-15217.7815
C00541=72.291,-9.737,87.405,177.2497,0.3746,-15217.6711
C00542=80.844,-10.790,89.614,177.4912,0.3380,-15217.6022
C00543=88.455,-11.935,90.663,177.9037,0.6505,-15217.6844
C00544=93.978,-15.553,91.206,179.1518,0.9927,-15219.3971
C00545=96.677,-21.285,91.642,179.8999,0.5802,-15222.4165
C00546=96.017,-27.936,92.077,-179.9899,0.0347,-15226.2223
C00547=93.742,-34.820,92.362,-179.9986,0.0037,-15230.3773
C00548=90.907,-41.664,92.362,-179.9983,0.0036,-15234.6227
C00549=87.648,-48.140,92.077,-179.9826,0.0317,-15238.7775
C00550=83.412,-53.310,91.642,-179.5190,0.3395,-15242.5833
C00551=77.451,-55.455,91.206,-178.6984,0.1022,-15245.6027
C00552=70.986,-54.108,90.663,-178.0578,-1.0228,-15247.3159
C00553=64.795,-49.536,89.614,-177.9867,-1.5357,-15247.3980
C00554=58.003,-44.233,87.405,-177.7900,-1.6809,-15247.3291
C00555=51.604,-39.197,84.354,-177.7091,-1.7240,-15247.2193
C00556=46.514,-35.238,81.229,-178.2854,-1.2476,-15247.1468
C00557=42.854,-33.363,78.888,167.1173,0.8020,-15247.9017
C00558=39.935,-34.660,77.945,159.3433,-15.7923,-15250.9551
C00559=38.350,-36.262,77.904,161.3555,-19.8142,-15253.3970
C00560=37.314,-37.314,77.932,160.7704,-19.2305,-15255.0000
C00561=36.262,-38.350,77.904,160.1853,-18.6440,-15256.6030
C00562=34.660,-39.935,77.945,164.2100,-20.6574,-15259.0449
C00563=33.363,-42.854,78.888,-179.1976,-12.8819,-15262.0983
C00564=35.238,-46.514,81.229,178.7524,1.7146,-15262.8532
C00565=39.197,-51.604,84.354,178.2760,2.2909,-15262.7807
C00566=44.233,-58.003,87.405,178.3191,2.2100,-15262.6709
C00567=49.536,-64.795,89.614,178.4643,2.0133,-15262.6020
C00568=54.108,-70.986,90.663,178.9772,1.9422,-15262.6841
C00569=55.455,-77.451,91.206,-179.8978,1.3016,-15264.3973
C00570=53.310,-83.412,91.642,-179.6605,0.4810,-15267.4167
C00571=48.140,-87.648,92.077,-179.9683,0.0174,-15271.2225
C00572=41.664,-90.907,92.362,-179.9964,0.0017,-15275.3773
C00573=34.820,-93.742,92.362,-179.9963,0.0014,-15279.6227
C00574=27.936,-96.017,92.077,-179.9653,0.0101,-15283.7777
C00575=21.285,-96.677,91.642,-179.4198,-0.1001,-15287.5835
C00576=15.553,-93.978,91.206,-179.0073,-0.8482,-15290.6029
C00577=11.935,-88.455,90.663,-179.3495,-2.0963,-15292.3156
C00578=10.790,-80.844,89.614,-179.6620,-2.5088,-15292.3978
C00579=9.737,-72.291,87.405,-179.6254,-2.7503,-15292.3289
C00580=8.774,-64.206,84.354,-179.5987,-2.8379,-15292.2185
C00581=7.974,-57.808,81.229,-179.6695,-2.0942,-15292.1462
C00582=6.711,-53.894,78.888,171.3670,9.7384,-15292.9019
C00583=3.730,-52.747,77.945,154.9876,3.8100,-15295.9551
C00584=1.476,-52.759,77.904,153.7405,-0.9277,-15298.3975
C00585=0.000,-52.771,77.932,153.7423,-0.0007,-15300.0000
C00586=0.000,-52.771,77.932,153.7423,-0.0007,-15300.0000
C00587=-1.476,-52.759,77.904,153.7405,0.9284,-15301.6025
C00588=-3.730,-52.747,77.945,154.9886,-3.8123,-15304.0449
C00589=-6.711,-53.894,78.888,171.3677,-9.7381,-15307.0981
C00590=-7.974,-57.808,81.229,-179.6695,2.0942,-15307.8538
C00591=-8.774,-64.206,84.354,-179.5987,2.8379,-15307.7815
C00592=-9.737,-72.291,87.405,-179.6254,2.7503,-15307.6711
C00593=-10.790,-80.844,89.614,-179.6620,2.5088,-15307.6022
C00594=-11.935,-88.455,90.663,-179.3495,2.0963,-15307.6844
C00595=-15.553,-93.978,91.206,-179.0073,0.8482,-15309.3971
C00596=-21.285,-96.677,91.642,-179.4198,0.1001,-15312.4165
C00597=-27.936,-96.017,92.077,-179.9653,-0.0101,-15316.2223
C00598=-34.820,-93.742,92.362,-179.9963,-0.0014,-15320.3773
C00599=-41.664,-90.907,92.362,-179.9964,-0.0017,-15324.6227
C00600=-48.140,-87.648,92.077,-179.9683,-0.0174,-15328.7775
C00601=-53.310,-83.412,91.642,-179.6605,-0.4810,-15332.5833
C00602=-55.455,-77.451,91.206,-179.8978,-1.3016,-15335.6027
C00603=-54.108,-70.986,90.663,178.9772,-1.9422,-15337.3159
C00604=-49.536,-64.795,89.614,178.4643,-2.0133,-15337.3980
C00605=-44.233,-58.003,87.405,178.3191,-2.2100,-15337.3291
C00606=-39.197,-51.604,84.354,178.2760,-2.2909,-15337.2193
C00607=-35.238,-46.514,81.229,178.7524,-1.7146,-15337.1468
C00608=-33.363,-42.854,78.888,-179.1980,12.8827,-15337.9017
C00609=-34.660,-39.935,77.945,164.2077,20.6567,-15340.9551
C00610=-36.262,-38.350,77.904,160.1858,18.6445,-15343.3970
C00611=-37.314,-37.314,77.932,160.7695,19.2296,-15345.0000
C00612=-38.350,-36.262,77.904,161.3560,19.8147,-15346.6030
C00613=-39.935,-34.660,77.945,159.3426,15.7900,-15349.0449
C00614=-42.854,-33.363,78.888,167.1181,-0.8024,-15352.0983
C00615=-46.514,-35.238,81.229,-178.2854,1.2476,-15352.8532
C00616=-51.604,-39.197,84.354,-177.7091,1.7240,-15352.7807
C00617=-58.003,-44.233,87.405,-177.7900,1.6809,-15352.6709
C00618=-64.795,-49.536,89.614,-177.9867,1.5357,-15352.6020
C00619=-70.986,-54.108,90.663,-178.0578,1.0228,-15352.6841
C00620=-77.451,-55.455,91.206,-178.6984,-0.1022,-15354.3973
C00621=-83.412,-53.310,91.642,-179.5190,-0.3395,-15357.4167
C00622=-87.648,-48.140,92.077,-179.9826,-0.0317,-15361.2225
C00623=-90.907,-41.664,92.362,-179.9983,-0.0036,-15365.3773
C00624=-93.742,-34.820,92.362,-179.9986,-0.0037,-15369.6227
C00625=-96.017,-27.936,92.077,-179.9899,-0.0347,-15373.7777
C00626=-96.677,-21.285,91.642,179.8999,-0.5802,-15377.5835
C00627=-93.978,-15.553,91.206,179.1518,-0.9927,-15380.6029
C00628=-88.455,-11.935,90.663,177.9037,-0.6505,-15382.3156
C00629=-80.844,-10.790,89.614,177.4912,-0.3380,-15382.3978
C00630=-72.291,-9.737,87.405,177.2497,-0.3746,-15382.3289
C00631=-64.206,-8.774,84.354,177.1621,-0.4013,-15382.2185
C00632=-57.808,-7.974,81.229,177.9058,-0.3305,-15382.1462
C00633=-53.894,-6.711,78.888,-170.2616,8.6330,-15382.9019
C00634=-52.747,-3.730,77.945,-176.1900,25.0124,-15385.9551
C00635=-52.759,-1.476,77.904,179.0723,26.2595,-15388.3975
C00636=-52.771,0.000,77.932,179.9993,26.2577,-15390.0000
C00637=-52.759,1.476,77.904,-179.0716,26.2595,-15391.6025
C00638=-52.747,3.730,77.945,176.1877,25.0114,-15394.0449
C00639=-53.894,6.711,78.888,170.2619,8.6323,-15397.0981
C00640=-57.808,7.974,81.229,-177.9058,-0.3305,-15397.8538
C00641=-64.206,8.774,84.354,-177.1621,-0.4013,-15397.7815
C00642=-72.291,9.737,87.405,-177.2497,-0.3746,-15397.6711
C00643=-80.844,10.790,89.614,-177.4912,-0.3380,-15397.6022
C00644=-88.455,11.935,90.663,-177.9037,-0.6505,-15397.6844
C00645=-93.978,15.553,91.206,-179.1518,-0.9927,-15399.3971
C00646=-96.677,21.285,91.642,-179.8999,-0.5802,-15402.4165
C00647=-96.017,27.936,92.077,179.9899,-0.0347,-15406.2223
C00648=-93.742,34.820,92.362,179.9986,-0.0037,-15410.3773
C00649=-90.907,41.664,92.362,179.9983,-0.0036,-15414.6227
C00650=-87.648,48.140,92.077,179.9826,-0.0317,-15418.7775
C00651=-83.412,53.310,91.642,179.5190,-0.3395,-15422.5833
C00652=-77.451,55.455,91.206,178.6984,-0.1022,-15425.6027
C00653=-70.986,54.108,90.663,178.0578,1.0228,-15427.3159
C00654=-64.795,49.536,89.614,177.9867,1.5357,-15427.3980
C00655=-58.003,44.233,87.405,177.7900,1.6809,-15427.3291
C00656=-51.604,39.197,84.354,177.7091,1.7240,-15427.2193
C00657=-46.514,35.238,81.229,178.2854,1.2476,-15427.1468
C00658=-42.854,33.363,78.888,-167.1173,-0.8020,-15427.9017
C00659=-39.935,34.660,77.945,-159.3433,15.7923,-15430.9551
C00660=-38.350,36.262,77.904,-161.3555,19.8142,-15433.3970
C00661=-37.314,37.314,77.932,-160.7704,19.2305,-15435.0000
C00662=-36.262,38.350,77.904,-160.1853,18.6440,-15436.6030
C00663=-34.660,39.935,77.945,-164.2100,20.6574,-15439.0449
C00664=-33.363,42.854,78.888,179.1976,12.8819,-15442.0983
C00665=-35.238,46.514,81.229,-178.7524,-1.7146,-15442.8532
C00666=-39.197,51.604,84.354,-178.2760,-2.2909,-15442.7807
C00667=-44.233,58.003,87.405,-178.3191,-2.2100,-15442.6709
C00668=-49.536,64.795,89.614,-178.4643,-2.0133,-15442.6020
C00669=-54.108,70.986,90.663,-178.9772,-1.9422,-15442.6841
C00670=-55.455,77.451,91.206,179.8978,-1.3016,-15444.3973
C00671=-53.310,83.412,91.642,179.6605,-0.4810,-15447.4167
C00672=-48.140,87.648,92.077,179.9683,-0.0174,-15451.2225
C00673=-41.664,90.907,92.362,179.9964,-0.0017,-15455.3773
C00674=-34.820,93.742,92.362,179.9963,-0.0014,-15459.6227
C00675=-27.936,96.017,92.077,179.9653,-0.0101,-15463.7777
C00676=-21.285,96.677,91.642,179.4198,0.1001,-15467.5835
C00677=-15.553,93.978,91.206,179.0073,0.8482,-15470.6029
C00678=-11.935,88.455,90.663,179.3495,2.0963,-15472.3156
C00679=-10.790,80.844,89.614,179.6620,2.5088,-15472.3978
C00680=-9.737,72.291,87.405,179.6254,2.7503,-15472.3289
C00681=-8.774,64.206,84.354,179.5987,2.8379,-15472.2185
C00682=-7.974,57.808,81.229,179.6695,2.0942,-15472.1462
C00683=-6.711,53.894,78.888,-171.3677,-9.7381,-15472.9019
C00684=-3.730,52.747,77.945,-154.9886,-3.8123,-15475.9551
C00685=-1.476,52.759,77.904,-153.7405,0.9284,-15478.3975
C00686=0.000,52.771,77.932,-153.7423,-0.0007,-15480.0000
C00687=0.000,51.832,79.921,-155.8023,-0.0006,-15480.0000
C00688=1.391,51.822,79.893,-155.7966,-0.7969,-15481.5376
C00689=3.586,51.820,79.935,-157.0572,3.6693,-15483.9586
C00690=6.543,53.038,80.908,-172.5244,8.6955,-15487.0327
C00691=7.793,57.125,83.313,179.7036,-1.9641,-15487.7683
C00692=8.610,63.749,86.500,179.6672,-2.4084,-15487.6919
C00693=9.608,72.041,89.587,179.7163,-2.1143,-15487.5966
C00694=10.692,80.728,91.809,179.7750,-1.6915,-15487.5446
C00695=11.850,88.408,92.861,179.6101,-1.2664,-15487.6343
C00696=15.484,93.970,93.405,179.4490,-0.4726,-15489.3569
C00697=21.237,96.685,93.841,179.7050,-0.0512,-15492.3884
C00698=27.910,96.026,94.277,179.9843,0.0045,-15496.2065
C00699=34.811,93.745,94.562,179.9985,0.0006,-15500.3718
C00700=41.672,90.903,94.562,179.9985,0.0007,-15504.6278
C00701=48.166,87.636,94.277,179.9857,0.0079,-15508.7938
C00702=53.350,83.383,93.841,179.8276,0.2448,-15512.6119
C00703=55.498,77.395,93.405,179.9446,0.7238,-15515.6434
C00704=54.135,70.893,92.861,-179.3801,1.1712,-15517.3659
C00705=49.523,64.644,91.809,-178.9628,1.3552,-15517.4553
C00706=44.146,57.735,89.587,-178.7052,1.6958,-15517.4027
C00707=38.990,51.166,86.500,-178.5316,1.9386,-15517.3085
C00708=34.883,45.903,83.313,-178.8204,1.5986,-15517.2322
C00709=32.877,42.130,80.908,179.1200,-11.3613,-15517.9674
C00710=34.107,39.178,79.935,-165.7499,-19.0172,-15521.0417
C00711=35.661,37.627,79.893,-161.8574,-17.1189,-15523.4634
C00712=36.651,36.651,79.921,-162.3718,-17.6274,-15525.0000
C00713=37.627,35.661,79.893,-162.8815,-18.1429,-15526.5366
C00714=39.178,34.107,79.935,-160.9822,-14.2479,-15528.9583
C00715=42.130,32.877,80.908,-168.6394,0.8803,-15532.0326
C00716=45.903,34.883,83.313,178.4014,-1.1796,-15532.7678
C00717=51.166,38.990,86.500,178.0614,-1.4684,-15532.6915
C00718=57.735,44.146,89.587,178.3042,-1.2948,-15532.5973
C00719=64.644,49.523,91.809,178.6448,-1.0372,-15532.5447
C00720=70.893,54.135,92.861,178.8288,-0.6199,-15532.6341
C00721=77.395,55.498,93.405,179.2762,0.0554,-15534.3566
C00722=83.383,53.350,93.841,179.7552,0.1724,-15537.3881
C00723=87.636,48.166,94.277,179.9921,0.0143,-15541.2062
C00724=90.903,41.672,94.562,179.9993,0.0015,-15545.3722
C00725=93.745,34.811,94.562,179.9994,0.0015,-15549.6282
C00726=96.026,27.910,94.277,179.9955,0.0157,-15553.7935
C00727=96.685,21.237,93.841,-179.9488,0.2950,-15557.6116
C00728=93.970,15.484,93.405,-179.5274,0.5510,-15560.6431
C00729=88.408,11.850,92.861,-178.7336,0.3899,-15562.3657
C00730=80.728,10.692,91.809,-178.3085,0.2250,-15562.4554
C00731=72.041,9.608,89.587,-177.8857,0.2837,-15562.4034
C00732=63.749,8.610,86.500,-177.5916,0.3328,-15562.3081
C00733=57.125,7.793,83.313,-178.0359,0.2964,-15562.2317
C00734=53.038,6.543,80.908,171.3045,-7.4756,-15562.9673
C00735=51.820,3.586,79.935,176.3307,-22.9428,-15566.0414
C00736=51.822,1.391,79.893,-179.2031,-24.2034,-15568.4624
C00737=51.832,0.000,79.921,-179.9994,-24.1977,-15570.0000
C00738=51.822,-1.390,79.893,179.2025,-24.2034,-15571.5365
C00739=51.820,-3.586,79.935,-176.3285,-22.9418,-15573.9586
C00740=53.038,-6.543,80.908,-171.3048,-7.4749,-15577.0327
C00741=57.125,-7.793,83.313,178.0359,0.2964,-15577.7683
C00742=63.749,-8.610,86.500,177.5916,0.3328,-15577.6919
C00743=72.041,-9.608,89.587,177.8857,0.2837,-15577.5966
C00744=80.728,-10.692,91.809,178.3085,0.2250,-15577.5446
C00745=88.408,-11.850,92.861,178.7336,0.3899,-15577.6343
C00746=93.970,-15.484,93.405,179.5274,0.5510,-15579.3569
C00747=96.685,-21.237,93.841,179.9488,0.2950,-15582.3884
C00748=96.026,-27.910,94.277,-179.9955,0.0157,-15586.2065
C00749=93.745,-34.811,94.562,-179.9994,0.0015,-15590.3718
C00750=90.903,-41.672,94.562,-179.9993,0.0015,-15594.6278
C00751=87.636,-48.166,94.277,-179.9921,0.0143,-15598.7938
C00752=83.383,-53.350,93.841,-179.7552,0.1724,-15602.6119
C00753=77.395,-55.498,93.405,-179.2762,0.0554,-15605.6434
C00754=70.893,-54.135,92.861,-178.8288,-0.6199,-15607.3659
C00755=64.644,-49.523,91.809,-178.6448,-1.0372,-15607.4553
C00756=57.735,-44.146,89.587,-178.3042,-1.2948,-15607.4027
C00757=51.166,-38.990,86.500,-178.0614,-1.4684,-15607.3085
C00758=45.903,-34.883,83.313,-178.4014,-1.1796,-15607.2322
C00759=42.130,-32.877,80.908,168.6387,0.8800,-15607.9674
C00760=39.178,-34.107,79.935,160.9828,-14.2501,-15611.0417
C00761=37.627,-35.661,79.893,162.8811,-18.1426,-15613.4634
C00762=36.651,-36.651,79.921,162.3726,-17.6282,-15615.0000
C00763=35.661,-37.627,79.893,161.8571,-17.1185,-15616.5366
C00764=34.107,-39.178,79.935,165.7521,-19.0178,-15618.9583
C00765=32.877,-42.130,80.908,-179.1197,-11.3606,-15622.0326
C00766=34.883,-45.903,83.313,178.8204,1.5986,-15622.7678
C00767=38.990,-51.166,86.500,178.5316,1.9386,-15622.6915
C00768=44.146,-57.735,89.587,178.7052,1.6958,-15622.5973
C00769=49.523,-64.644,91.809,178.9628,1.3552,-15622.5447
C00770=54.135,-70.893,92.861,179.3801,1.1712,-15622.6341
C00771=55.498,-77.395,93.405,-179.9446,0.7238,-15624.3566
C00772=53.350,-83.383,93.841,-179.8276,0.2448,-15627.3881
C00773=48.166,-87.636,94.277,-179.9857,0.0079,-15631.2062
C00774=41.672,-90.903,94.562,-179.9985,0.0007,-15635.3722
C00775=34.811,-93.745,94.562,-179.9985,0.0006,-15639.6282
C00776=27.910,-96.026,94.277,-179.9843,0.0045,-15643.7935
C00777=21.237,-96.685,93.841,-179.7050,-0.0512,-15647.6116
C00778=15.484,-93.970,93.405,-179.4490,-0.4726,-15650.6431
C00779=11.850,-88.408,92.861,-179.6101,-1.2664,-15652.3657
C00780=10.692,-80.728,91.809,-179.7750,-1.6915,-15652.4554
C00781=9.608,-72.041,89.587,-179.7163,-2.1143,-15652.4034
C00782=8.610,-63.749,86.500,-179.6672,-2.4084,-15652.3081
C00783=7.793,-57.125,83.313,-179.7036,-1.9641,-15652.2317
C00784=6.543,-53.038,80.908,172.5244,8.6955,-15652.9673
C00785=3.586,-51.820,79.935,157.0572,3.6693,-15656.0414
C00786=1.391,-51.822,79.893,155.7966,-0.7969,-15658.4624
C00787=0.000,-51.832,79.921,155.8023,-0.0006,-15660.0000
C00788=0.000,-51.832,79.921,155.8023,-0.0006,-15660.0000
C00789=-1.390,-51.822,79.893,155.7966,0.7975,-15661.5365
C00790=-3.586,-51.820,79.935,157.0582,-3.6715,-15663.9586
C00791=-6.543,-53.038,80.908,172.5251,-8.6952,-15667.0327
C00792=-7.793,-57.125,83.313,-179.7036,1.9641,-15667.7683
C00793=-8.610,-63.749,86.500,-179.6672,2.4084,-15667.6919
C00794=-9.608,-72.041,89.587,-179.7163,2.1143,-15667.5966
C00795=-10.692,-80.728,91.809,-179.7750,1.6915,-15667.5446
C00796=-11.850,-88.408,92.861,-179.6101,1.2664,-15667.6343
C00797=-15.484,-93.970,93.405,-179.4490,0.4726,-15669.3569
C00798=-21.237,-96.685,93.841,-179.7050,0.0512,-15672.3884
C00799=-27.910,-96.026,94.277,-179.9843,-0.0045,-15676.2065
C00800=-34.811,-93.745,94.562,-179.9985,-0.0006,-15680.3718
C00801=-41.672,-90.903,94.562,-179.9985,-0.0007,-15684.6278
C00802=-48.166,-87.636,94.277,-179.9857,-0.0079,-15688.7938
C00803=-53.350,-83.383,93.841,-179.8276,-0.2448,-15692.6119
C00804=-55.498,-77.395,93.405,-179.9446,-0.7238,-15695.6434
C00805=-54.135,-70.893,92.861,179.3801,-1.1712,-15697.3659
C00806=-49.523,-64.644,91.809,178.9628,-1.3552,-15697.4553
C00807=-44.146,-57.735,89.587,178.7052,-1.6958,-15697.4027
C00808=-38.990,-51.166,86.500,178.5316,-1.9386,-15697.3085
C00809=-34.883,-45.903,83.313,178.8204,-1.5986,-15697.2322
C00810=-32.877,-42.130,80.908,-179.1200,11.3613,-15697.9674
C00811=-34.107,-39.178,79.935,165.7499,19.0172,-15701.0417
C00812=-35.661,-37.627,79.893,161.8574,17.1189,-15703.4634
C00813=-36.651,-36.651,79.921,162.3718,17.6274,-15705.0000
C00814=-37.627,-35.661,79.893,162.8815,18.1429,-15706.5366
C00815=-39.178,-34.107,79.935,160.9822,14.2479,-15708.9583
C00816=-42.130,-32.877,80.908,168.6394,-0.8803,-15712.0326
C00817=-45.903,-34.883,83.313,-178.4014,1.1796,-15712.7678
C00818=-51.166,-38.990,86.500,-178.0614,1.4684,-15712.6915
C00819=-57.735,-44.146,89.587,-178.3042,1.2948,-15712.5973
C00820=-64.644,-49.523,91.809,-178.6448,1.0372,-15712.5447
C00821=-70.893,-54.135,92.861,-178.8288,0.6199,-15712.6341
C00822=-77.395,-55.498,93.405,-179.2762,-0.0554,-15714.3566
C00823=-83.383,-53.350,93.841,-179.7552,-0.1724,-15717.3881
C00824=-87.636,-48.166,94.277,-179.9921,-0.0143,-15721.2062
C00825=-90.903,-41.672,94.562,-179.9993,-0.0015,-15725.3722
C00826=-93.745,-34.811,94.562,-179.9994,-0.0015,-15729.6282
C00827=-96.026,-27.910,94.277,-179.9955,-0.0157,-15733.7935
C00828=-96.685,-21.237,93.841,179.9488,-0.2950,-15737.6116
C00829=-93.970,-15.484,93.405,179.5274,-0.5510,-15740.6431
C00830=-88.408,-11.850,92.861,178.7336,-0.3899,-15742.3657
C00831=-80.728,-10.692,91.809,178.3085,-0.2250,-15742.4554
C00832=-72.041,-9.608,89.587,177.8857,-0.2837,-15742.4034
C00833=-63.749,-8.610,86.500,177.5916,-0.3328,-15742.3081
C00834=-57.125,-7.793,83.313,178.0359,-0.2964,-15742.2317
C00835=-53.038,-6.543,80.908,-171.3045,7.4756,-15742.9673
C00836=-51.820,-3.586,79.935,-176.3307,22.9428,-15746.0414
C00837=-51.822,-1.391,79.893,179.2031,24.2034,-15748.4624
C00838=-51.832,0.000,79.921,179.9994,24.1977,-15750.0000
C00839=-51.822,1.390,79.893,-179.2025,24.2034,-15751.5365
C00840=-51.820,3.586,79.935,176.3285,22.9418,-15753.9586
C00841=-53.038,6.543,80.908,171.3048,7.4749,-15757.0327
C00842=-57.125,7.793,83.313,-178.0359,-0.2964,-15757.7683
C00843=-63.749,8.610,86.500,-177.5916,-0.3328,-15757.6919
C00844=-72.041,9.608,89.587,-177.8857,-0.2837,-15757.5966
C00845=-80.728,10.692,91.809,-178.3085,-0.2250,-15757.5446
C00846=-88.408,11.850,92.861,-178.7336,-0.3899,-15757.6343
C00847=-93.970,15.484,93.405,-179.5274,-0.5510,-15759.3569
C00848=-96.685,21.237,93.841,-179.9488,-0.2950,-15762.3884
C00849=-96.026,27.910,94.277,179.9955,-0.0157,-15766.2065
C00850=-93.745,34.811,94.562,179.9994,-0.0015,-15770.3718
C00851=-90.903,41.672,94.562,179.9993,-0.0015,-15774.6278
C00852=-87.636,48.166,94.277,179.9921,-0.0143,-15778.7938
C00853=-83.383,53.350,93.841,179.7552,-0.1724,-15782.6119
C00854=-77.395,55.498,93.405,179.2762,-0.0554,-15785.6434
C00855=-70.893,54.135,92.861,178.8288,0.6199,-15787.3659
C00856=-64.644,49.523,91.809,178.6448,1.0372,-15787.4553
C00857=-57.735,44.146,89.587,178.3042,1.2948,-15787.4027
C00858=-51.166,38.990,86.500,178.0614,1.4684,-15787.3085
C00859=-45.903,34.883,83.313,178.4014,1.1796,-15787.2322
C00860=-42.130,32.877,80.908,-168.6387,-0.8800,-15787.9674
C00861=-39.178,34.107,79.935,-160.9828,14.2501,-15791.0417
C00862=-37.627,35.661,79.893,-162.8811,18.1426,-15793.4634
C00863=-36.651,36.651,79.921,-162.3726,17.6282,-15795.0000
C00864=-35.661,37.627,79.893,-161.8571,17.1185,-15796.5366
C00865=-34.107,39.178,79.935,-165.7521,19.0178,-15798.9583
C00866=-32.877,42.130,80.908,179.1197,11.3606,-15802.0326
C00867=-34.883,45.903,83.313,-178.8204,-1.5986,-15802.7678
C00868=-38.990,51.166,86.500,-178.5316,-1.9386,-15802.6915
C00869=-44.146,57.735,89.587,-178.7052,-1.6958,-15802.5973
C00870=-49.523,64.644,91.809,-178.9628,-1.3552,-15802.5447
C00871=-54.135,70.893,92.861,-179.3801,-1.1712,-15802.6341
C00872=-55.498,77.395,93.405,179.9446,-0.7238,-15804.3566
C00873=-53.350,83.383,93.841,179.8276,-0.2448,-15807.3881
C00874=-48.166,87.636,94.277,179.9857,-0.0079,-15811.2062
C00875=-41.672,90.903,94.562,179.9985,-0.0007,-15815.3722
C00876=-34.811,93.745,94.562,179.9985,-0.0006,-15819.6282
C00877=-27.910,96.026,94.277,179.9843,-0.0045,-15823.7935
C00878=-21.237,96.685,93.841,179.7050,0.0512,-15827.6116
C00879=-15.484,93.970,93.405,179.4490,0.4726,-15830.6431
C00880=-11.850,88.408,92.861,179.6101,1.2664,-15832.3657
C00881=-10.692,80.728,91.809,179.7750,1.6915,-15832.4554
C00882=-9.608,72.041,89.587,179.7163,2.1143,-15832.4034
C00883=-8.610,63.749,86.500,179.6672,2.4084,-15832.3081
C00884=-7.793,57.125,83.313,179.7036,1.9641,-15832.2317
C00885=-6.543,53.038,80.908,-172.5251,-8.6952,-15832.9673
C00886=-3.586,51.820,79.935,-157.0582,-3.6715,-15836.0414
C00887=-1.390,51.822,79.893,-155.7966,0.7975,-15838.4635
C00888=0.000,51.832,79.921,-155.8023,-0.0006,-15840.0000
C00889=0.000,50.970,81.946,-158.1022,-0.0005,-15840.0000
C00890=1.312,50.962,81.916,-158.0920,-0.6690,-15841.4747
C00891=3.453,50.970,81.960,-159.3373,3.4481,-15843.8756
C00892=6.389,52.261,82.960,-173.6406,7.6045,-15846.9699
C00893=7.633,56.525,85.423,179.7440,-1.7649,-15847.6906
C00894=8.475,63.374,88.663,179.7387,-1.9278,-15847.6170
C00895=9.515,71.858,91.777,179.8100,-1.4311,-15847.5429
C00896=10.634,80.658,94.007,179.8912,-0.8247,-15847.5106
C00897=11.808,88.386,95.061,179.8809,-0.3884,-15847.6094
C00898=15.455,93.966,95.604,179.9140,-0.0739,-15849.3401
C00899=55.516,77.372,95.604,179.9914,0.1131,-15875.6602
C00900=54.149,70.847,95.061,-179.8096,0.3589,-15877.3910
C00901=49.515,64.553,94.007,-179.4937,0.6602,-15877.4898
C00902=44.083,57.539,91.777,-179.1223,1.1463,-15877.4572
C00903=38.820,50.805,88.663,-178.8213,1.5481,-15877.3834
C00904=34.571,45.367,85.423,-178.9328,1.4291,-15877.3085
C00905=32.436,41.472,82.960,179.1064,-9.8268,-15878.0296
C00906=33.599,38.483,81.960,-167.3708,-17.1854,-15881.1238
C00907=35.108,36.963,81.916,-163.6891,-15.4355,-15883.5256
C00908=36.041,36.041,81.946,-164.1333,-15.8661,-15885.0000
C00909=36.963,35.108,81.916,-164.5648,-16.3112,-15886.4744
C00910=38.483,33.599,81.960,-162.8140,-12.6271,-15888.8762
C00911=41.472,32.436,82.960,-170.1739,0.8939,-15891.9704
C00912=45.367,34.571,85.423,178.5709,-1.0672,-15892.6915
C00913=50.805,38.820,88.663,178.4519,-1.1787,-15892.6166
C00914=57.539,44.083,91.777,178.8537,-0.8777,-15892.5428
C00915=64.553,49.515,94.007,179.3398,-0.5063,-15892.5102
C00916=70.847,54.149,95.061,179.6411,-0.1904,-15892.6090
C00917=77.372,55.516,95.604,179.8869,0.0086,-15894.3398
C00918=93.966,15.455,95.604,-179.9261,0.0860,-15920.6599
C00919=88.386,11.808,95.061,-179.6116,0.1191,-15922.3906
C00920=80.658,10.634,94.007,-179.1753,0.1088,-15922.4894
C00921=71.858,9.515,91.777,-178.5689,0.1900,-15922.4571
C00922=63.374,8.475,88.663,-178.0722,0.2613,-15922.3830
C00923=56.525,7.633,85.423,-178.2351,0.2560,-15922.3094
C00924=52.261,6.389,82.960,172.3955,-6.3594,-15923.0301
C00925=50.970,3.453,81.960,176.5519,-20.6627,-15926.1244
C00926=50.962,1.312,81.916,-179.3310,-21.9080,-15928.5253
C00927=50.970,0.000,81.946,-179.9995,-21.8978,-15930.0000
C00928=50.962,-1.311,81.916,179.3306,-21.9080,-15931.4736
C00929=50.970,-3.454,81.960,-176.5499,-20.6618,-15933.8767
C00930=52.261,-6.389,82.960,-172.3958,-6.3587,-15936.9699
C00931=56.525,-7.633,85.423,178.2351,0.2560,-15937.6906
C00932=63.374,-8.475,88.663,178.0722,0.2613,-15937.6170
C00933=71.858,-9.515,91.777,178.5689,0.1900,-15937.5429
C00934=80.658,-10.634,94.007,179.1753,0.1088,-15937.5106
C00935=88.386,-11.808,95.061,179.6116,0.1191,-15937.6094
C00936=93.966,-15.455,95.604,179.9261,0.0860,-15939.3401
C00937=77.372,-55.516,95.604,-179.8869,0.0086,-15965.6602
C00938=70.847,-54.149,95.061,-179.6411,-0.1904,-15967.3910
C00939=64.553,-49.515,94.007,-179.3398,-0.5063,-15967.4898
C00940=57.539,-44.083,91.777,-178.8537,-0.8777,-15967.4572
C00941=50.805,-38.820,88.663,-178.4519,-1.1787,-15967.3834
C00942=45.367,-34.571,85.423,-178.5709,-1.0672,-15967.3085
C00943=41.472,-32.436,82.960,170.1732,0.8936,-15968.0296
C00944=38.483,-33.599,81.960,162.8146,-12.6292,-15971.1238
C00945=36.963,-35.108,81.916,164.5645,-16.3109,-15973.5256
C00946=36.041,-36.041,81.946,164.1339,-15.8667,-15975.0000
C00947=35.108,-36.963,81.916,163.6888,-15.4352,-15976.4744
C00948=33.599,-38.483,81.960,167.3729,-17.1860,-15978.8762
C00949=32.436,-41.472,82.960,-179.1061,-9.8261,-15981.9704
C00950=34.571,-45.367,85.423,178.9328,1.4291,-15982.6915
C00951=38.820,-50.805,88.663,178.8213,1.5481,-15982.6166
C00952=44.083,-57.539,91.777,179.1223,1.1463,-15982.5428
C00953=49.515,-64.553,94.007,179.4937,0.6602,-15982.5102
C00954=54.149,-70.847,95.061,179.8096,0.3589,-15982.6090
C00955=55.516,-77.372,95.604,-179.9914,0.1131,-15984.3398
C00956=15.455,-93.966,95.604,-179.9140,-0.0739,-16010.6599
C00957=11.808,-88.386,95.061,-179.8809,-0.3884,-16012.3906
C00958=10.634,-80.658,94.007,-179.8912,-0.8247,-16012.4894
C00959=9.515,-71.858,91.777,-179.8100,-1.4311,-16012.4571
C00960=8.475,-63.374,88.663,-179.7387,-1.9278,-16012.3830
C00961=7.633,-56.525,85.423,-179.7440,-1.7649,-16012.3094
C00962=6.389,-52.261,82.960,173.6406,7.6045,-16013.0301
C00963=3.453,-50.970,81.960,159.3373,3.4481,-16016.1244
C00964=1.312,-50.962,81.916,158.0920,-0.6690,-16018.5253
C00965=0.000,-50.970,81.946,158.1022,-0.0005,-16020.0000
C00966=0.000,-50.970,81.946,158.1022,-0.0005,-16020.0000
C00967=-1.311,-50.962,81.916,158.0920,0.6694,-16021.4736
C00968=-3.454,-50.970,81.960,159.3382,-3.4501,-16023.8767
C00969=-6.389,-52.261,82.960,173.6413,-7.6042,-16026.9699
C00970=-7.633,-56.525,85.423,-179.7440,1.7649,-16027.6906
C00971=-8.475,-63.374,88.663,-179.7387,1.9278,-16027.6170
C00972=-9.515,-71.858,91.777,-179.8100,1.4311,-16027.5429
C00973=-10.634,-80.658,94.007,-179.8912,0.8247,-16027.5106
C00974=-11.808,-88.386,95.061,-179.8809,0.3884,-16027.6094
C00975=-15.455,-93.966,95.604,-179.9140,0.0739,-16029.3401
C00976=-55.516,-77.372,95.604,-179.9914,-0.1131,-16055.6602
C00977=-54.149,-70.847,95.061,179.8096,-0.3589,-16057.3910
C00978=-49.515,-64.553,94.007,179.4937,-0.6602,-16057.4898
C00979=-44.083,-57.539,91.777,179.1223,-1.1463,-16057.4572
C00980=-38.820,-50.805,88.663,178.8213,-1.5481,-16057.3834
C00981=-34.571,-45.367,85.423,178.9328,-1.4291,-16057.3085
C00982=-32.436,-41.472,82.960,-179.1064,9.8268,-16058.0296
C00983=-33.599,-38.483,81.960,167.3708,17.1854,-16061.1238
C00984=-35.108,-36.963,81.916,163.6891,15.4355,-16063.5256
C00985=-36.041,-36.041,81.946,164.1333,15.8661,-16065.0000
C00986=-36.963,-35.108,81.916,164.5648,16.3112,-16066.4744
C00987=-38.483,-33.599,81.960,162.8140,12.6271,-16068.8762
C00988=-41.472,-32.436,82.960,170.1739,-0.8939,-16071.9704
C00989=-45.367,-34.571,85.423,-178.5709,1.0672,-16072.6915
C00990=-50.805,-38.820,88.663,-178.4519,1.1787,-16072.6166
C00991=-57.539,-44.083,91.777,-178.8537,0.8777,-16072.5428
C00992=-64.553,-49.515,94.007,-179.3398,0.5063,-16072.5102
C00993=-70.847,-54.149,95.061,-179.6411,0.1904,-16072.6090
C00994=-77.372,-55.516,95.604,-179.8869,-0.0086,-16074.3398
C00995=-93.966,-15.455,95.604,179.9261,-0.0860,-16100.6599
C00996=-88.386,-11.808,95.061,179.6116,-0.1191,-16102.3906
C00997=-80.658,-10.634,94.007,179.1753,-0.1088,-16102.4894
C00998=-71.858,-9.515,91.777,178.5689,-0.1900,-16102.4571
C00999=-63.374,-8.475,88.663,178.0722,-0.2613,-16102.3830
C01000=-56.525,-7.633,85.423,178.2351,-0.2560,-16102.3094
C01001=-52.261,-6.389,82.960,-172.3955,6.3594,-16103.0301
C01002=-50.970,-3.453,81.960,-176.5519,20.6627,-16106.1244
C01003=-50.962,-1.312,81.916,179.3310,21.9080,-16108.5253
C01004=-50.970,0.000,81.946,179.9995,21.8978,-16110.0000
C01005=-50.962,1.311,81.916,-179.3306,21.9080,-16111.4736
C01006=-50.970,3.454,81.960,176.5499,20.6618,-16113.8767
C01007=-52.261,6.389,82.960,172.3958,6.3587,-16116.9699
C01008=-56.525,7.633,85.423,-178.2351,-0.2560,-16117.6906
C01009=-63.374,8.475,88.663,-178.0722,-0.2613,-16117.6170
C01010=-71.858,9.515,91.777,-178.5689,-0.1900,-16117.5429
C01011=-80.658,10.634,94.007,-179.1753,-0.1088,-16117.5106
C01012=-88.386,11.808,95.061,-179.6116,-0.1191,-16117.6094
C01013=-93.966,15.455,95.604,-179.9261,-0.0860,-16119.3401
C01014=-77.372,55.516,95.604,179.8869,-0.0086,-16145.6602
C01015=-70.847,54.149,95.061,179.6411,0.1904,-16147.3910
C01016=-64.553,49.515,94.007,179.3398,0.5063,-16147.4898
C01017=-57.539,44.083,91.777,178.8537,0.8777,-16147.4572
C01018=-50.805,38.820,88.663,178.4519,1.1787,-16147.3834
C01019=-45.367,34.571,85.423,178.5709,1.0672,-16147.3085
C01020=-41.472,32.436,82.960,-170.1732,-0.8936,-16148.0296
C01021=-38.483,33.599,81.960,-162.8146,12.6292,-16151.1238
C01022=-36.963,35.108,81.916,-164.5645,16.3109,-16153.5256
C01023=-36.041,36.041,81.946,-164.1339,15.8667,-16155.0000
C01024=-35.108,36.963,81.916,-163.6888,15.4352,-16156.4744
C01025=-33.599,38.483,81.960,-167.3729,17.1860,-16158.8762
C01026=-32.436,41.472,82.960,179.1061,9.8261,-16161.9704
C01027=-34.571,45.367,85.423,-178.9328,-1.4291,-16162.6915
C01028=-38.820,50.805,88.663,-178.8213,-1.5481,-16162.6166
C01029=-44.083,57.539,91.777,-179.1223,-1.1463,-16162.5428
C01030=-49.515,64.553,94.007,-179.4937,-0.6602,-16162.5102
C01031=-54.149,70.847,95.061,-179.8096,-0.3589,-16162.6090
C01032=-55.516,77.372,95.604,179.9914,-0.1131,-16164.3398
C01033=-15.455,93.966,95.604,179.9140,0.0739,-16190.6599
C01034=-11.808,88.386,95.061,179.8809,0.3884,-16192.3906
C01035=-10.634,80.658,94.007,179.8912,0.8247,-16192.4894
C01036=-9.515,71.858,91.777,179.8100,1.4311,-16192.4571
C01037=-8.475,63.374,88.663,179.7387,1.9278,-16192.3830
C01038=-7.633,56.525,85.423,179.7440,1.7649,-16192.3094
C01039=-6.389,52.261,82.960,-173.6413,-7.6042,-16193.0301
C01040=-3.454,50.970,81.960,-159.3382,-3.4501,-16196.1233
C01041=-1.311,50.962,81.916,-158.0920,0.6694,-16198.5264
C01042=0.000,50.970,81.946,-158.1022,-0.0005,-16200.0000
C01043=0.000,50.195,84.004,-160.6619,-0.0004,-16200.0000
C01044=1.241,50.188,83.974,-160.6464,-0.5462,-16201.4165
C01045=3.334,50.204,84.019,-161.8405,3.1426,-16203.7994
C01046=6.253,51.571,85.045,-174.7212,6.4678,-16206.9134
C01047=7.499,56.017,87.559,179.7895,-1.5010,-16207.6249
C01048=8.371,63.087,90.842,179.8130,-1.3996,-16207.5584
C01049=9.459,71.748,93.974,179.9071,-0.7043,-16207.5104
C01050=44.045,57.421,93.974,-179.5677,0.5637,-16237.4901
C01051=38.690,50.529,90.842,-179.1424,1.1219,-16237.4412
C01052=34.307,44.912,87.559,-179.0873,1.2103,-16237.3752
C01053=32.045,40.888,85.045,179.1504,-8.2781,-16238.0867
C01054=33.142,37.857,84.019,-169.0703,-15.1499,-16241.2006
C01055=34.611,36.365,83.974,-165.6885,-13.5839,-16243.5844
C01056=35.493,35.493,84.004,-166.0631,-13.9364,-16245.0000
C01057=36.365,34.611,83.974,-166.4163,-14.3116,-16246.4156
C01058=37.858,33.142,84.019,-164.8496,-10.9278,-16248.8001
C01059=40.888,32.045,85.045,-171.7226,0.8499,-16251.9133
C01060=44.912,34.307,87.559,178.7897,-0.9127,-16252.6248
C01061=50.529,38.690,90.842,178.8781,-0.8576,-16252.5588
C01062=57.421,44.045,93.974,179.4363,-0.4323,-16252.5099
C01063=71.748,9.459,93.974,-179.2957,0.0929,-16282.4896
C01064=63.087,8.371,90.842,-178.6004,0.1870,-16282.4416
C01065=56.017,7.499,87.559,-178.4990,0.2105,-16282.3751
C01066=51.571,6.253,85.045,173.5322,-5.2788,-16283.0866
C01067=50.204,3.334,84.019,176.8574,-18.1595,-16286.2006
C01068=50.188,1.241,83.974,-179.4538,-19.3536,-16288.5835
C01069=50.195,0.000,84.004,-179.9996,-19.3381,-16290.0000
C01070=50.188,-1.240,83.974,179.4535,-19.3536,-16291.4153
C01071=50.204,-3.335,84.019,-176.8556,-18.1586,-16293.8005
C01072=51.571,-6.253,85.045,-173.5325,-5.2781,-16296.9134
C01073=56.017,-7.499,87.559,178.4990,0.2105,-16297.6249
C01074=63.087,-8.371,90.842,178.6004,0.1870,-16297.5584
C01075=71.748,-9.459,93.974,179.2957,0.0929,-16297.5104
C01076=57.421,-44.045,93.974,-179.4363,-0.4323,-16327.4901
C01077=50.529,-38.690,90.842,-178.8781,-0.8576,-16327.4412
C01078=44.912,-34.307,87.559,-178.7897,-0.9127,-16327.3752
C01079=40.888,-32.045,85.045,171.7219,0.8496,-16328.0867
C01080=37.857,-33.142,84.019,164.8501,-10.9297,-16331.2006
C01081=36.365,-34.611,83.974,166.4161,-14.3115,-16333.5844
C01082=35.493,-35.493,84.004,166.0636,-13.9369,-16335.0000
C01083=34.611,-36.365,83.974,165.6884,-13.5837,-16336.4156
C01084=33.142,-37.858,84.019,169.0722,-15.1504,-16338.8001
C01085=32.045,-40.888,85.045,-179.1501,-8.2774,-16341.9133
C01086=34.307,-44.912,87.559,179.0873,1.2103,-16342.6248
C01087=38.690,-50.529,90.842,179.1424,1.1219,-16342.5588
C01088=44.045,-57.421,93.974,179.5677,0.5637,-16342.5099
C01089=9.459,-71.748,93.974,-179.9071,-0.7043,-16372.4896
C01090=8.371,-63.087,90.842,-179.8130,-1.3996,-16372.4416
C01091=7.499,-56.017,87.559,-179.7895,-1.5010,-16372.3751
C01092=6.253,-51.571,85.045,174.7212,6.4678,-16373.0866
C01093=3.334,-50.204,84.019,161.8405,3.1426,-16376.2006
C01094=1.241,-50.188,83.974,160.6464,-0.5462,-16378.5835
C01095=0.000,-50.195,84.004,160.6619,-0.0004,-16380.0000
C01096=0.000,-50.195,84.004,160.6619,-0.0004,-16380.0000
C01097=-1.240,-50.188,83.974,160.6464,0.5465,-16381.4153
C01098=-3.335,-50.204,84.019,161.8414,-3.1444,-16383.8005
C01099=-6.253,-51.571,85.045,174.7219,-6.4675,-16386.9134
C01100=-7.499,-56.017,87.559,-179.7895,1.5010,-16387.6249
C01101=-8.371,-63.087,90.842,-179.8130,1.3996,-16387.5584
C01102=-9.459,-71.748,93.974,-179.9071,0.7043,-16387.5104
C01103=-44.045,-57.421,93.974,179.5677,-0.5637,-16417.4901
C01104=-38.690,-50.529,90.842,179.1424,-1.1219,-16417.4412
C01105=-34.307,-44.912,87.559,179.0873,-1.2103,-16417.3752
C01106=-32.045,-40.888,85.045,-179.1504,8.2781,-16418.0867
C01107=-33.142,-37.857,84.019,169.0703,15.1499,-16421.2006
C01108=-34.611,-36.365,83.974,165.6885,13.5839,-16423.5844
C01109=-35.493,-35.493,84.004,166.0631,13.9364,-16425.0000
C01110=-36.365,-34.611,83.974,166.4163,14.3116,-16426.4156
C01111=-37.858,-33.142,84.019,164.8496,10.9278,-16428.8001
C01112=-40.888,-32.045,85.045,171.7226,-0.8499,-16431.9133
C01113=-44.912,-34.307,87.559,-178.7897,0.9127,-16432.6248
C01114=-50.529,-38.690,90.842,-178.8781,0.8576,-16432.5588
C01115=-57.421,-44.045,93.974,-179.4363,0.4323,-16432.5099
C01116=-71.748,-9.459,93.974,179.2957,-0.0929,-16462.4896
C01117=-63.087,-8.371,90.842,178.6004,-0.1870,-16462.4416
C01118=-56.017,-7.499,87.559,178.4990,-0.2105,-16462.3751
C01119=-51.571,-6.253,85.045,-173.5322,5.2788,-16463.0866
C01120=-50.204,-3.334,84.019,-176.8574,18.1595,-16466.2006
C01121=-50.188,-1.241,83.974,179.4538,19.3536,-16468.5835
C01122=-50.195,0.000,84.004,179.9996,19.3381,-16470.0000
C01123=-50.188,1.240,83.974,-179.4535,19.3536,-16471.4153
C01124=-50.204,3.335,84.019,176.8556,18.1586,-16473.8005
C01125=-51.571,6.253,85.045,173.5325,5.2781,-16476.9134
C01126=-56.017,7.499,87.559,-178.4990,-0.2105,-16477.6249
C01127=-63.087,8.371,90.842,-178.6004,-0.1870,-16477.5584
C01128=-71.748,9.459,93.974,-179.2957,-0.0929,-16477.5104
C01129=-57.421,44.045,93.974,179.4363,0.4323,-16507.4901
C01130=-50.529,38.690,90.842,178.8781,0.8576,-16507.4412
C01131=-44.912,34.307,87.559,178.7897,0.9127,-16507.3752
C01132=-40.888,32.045,85.045,-171.7219,-0.8496,-16508.0867
C01133=-37.857,33.142,84.019,-164.8501,10.9297,-16511.2006
C01134=-36.365,34.611,83.974,-166.4161,14.3115,-16513.5844
C01135=-35.493,35.493,84.004,-166.0636,13.9369,-16515.0000
C01136=-34.611,36.365,83.974,-165.6884,13.5837,-16516.4156
C01137=-33.142,37.858,84.019,-169.0722,15.1504,-16518.8001
C01138=-32.045,40.888,85.045,179.1501,8.2774,-16521.9133
C01139=-34.307,44.912,87.559,-179.0873,-1.2103,-16522.6248
C01140=-38.690,50.529,90.842,-179.1424,-1.1219,-16522.5588
C01141=-44.045,57.421,93.974,-179.5677,-0.5637,-16522.5099
C01142=-9.459,71.748,93.974,179.9071,0.7043,-16552.4896
C01143=-8.371,63.087,90.842,179.8130,1.3996,-16552.4416
C01144=-7.499,56.017,87.559,179.7895,1.5010,-16552.3751
C01145=-6.253,51.571,85.045,-174.7219,-6.4675,-16553.0866
C01146=-3.335,50.204,84.019,-161.8414,-3.1444,-16556.1995
C01147=-1.240,50.188,83.974,-160.6464,0.5465,-16558.5847
C01148=0.000,50.195,84.004,-160.6619,-0.0004,-16560.0000
C01149=0.000,49.517,86.097,-163.4981,-0.0002,-16560.0000
C01150=1.179,49.510,86.067,-163.4764,-0.4305,-16561.3641
C01151=3.230,49.536,86.112,-164.5770,2.7513,-16563.7307
C01152=6.137,50.981,87.161,-175.7739,5.2863,-16566.8641
C01153=7.391,55.610,89.719,179.8393,-1.1782,-16567.5707
C01154=8.302,62.896,93.033,179.8904,-0.8284,-16567.5193
C01155=38.603,50.345,93.033,-179.4917,0.6633,-16597.4799
C01156=34.096,44.548,89.719,-179.2805,0.9468,-16597.4296
C01157=31.710,40.389,87.161,179.2451,-6.7115,-16598.1360
C01158=32.743,37.311,86.112,-170.8486,-12.9014,-16601.2692
C01159=34.176,35.843,86.067,-167.8615,-11.5554,-16603.6362
C01160=35.014,35.014,86.097,-168.1686,-11.8311,-16605.0000
C01161=35.842,34.176,86.067,-168.4447,-12.1386,-16606.3630
C01162=37.311,32.743,86.112,-167.0982,-9.1497,-16608.7308
C01163=40.389,31.710,87.161,-173.2891,0.7551,-16611.8640
C01164=44.548,34.096,89.719,179.0532,-0.7195,-16612.5704
C01165=50.345,38.603,93.033,179.3367,-0.5083,-16612.5201
C01166=62.896,8.302,93.033,-179.1716,0.1096,-16642.4807
C01167=55.610,7.391,89.719,-178.8218,0.1607,-16642.4293
C01168=50.981,6.137,87.161,174.7137,-4.2261,-16643.1359
C01169=49.536,3.230,86.112,177.2487,-15.4230,-16646.2693
C01170=49.510,1.179,86.067,-179.5695,-16.5236,-16648.6359
C01171=49.517,0.000,86.097,-179.9998,-16.5019,-16650.0000
C01172=49.510,-1.178,86.067,179.5694,-16.5236,-16651.3630
C01173=49.536,-3.231,86.112,-177.2471,-15.4221,-16653.7318
C01174=50.981,-6.137,87.161,-174.7140,-4.2255,-16656.8641
C01175=55.610,-7.391,89.719,178.8218,0.1607,-16657.5707
C01176=62.896,-8.302,93.033,179.1716,0.1096,-16657.5193
C01177=50.345,-38.603,93.033,-179.3367,-0.5083,-16687.4799
C01178=44.548,-34.096,89.719,-179.0532,-0.7195,-16687.4296
C01179=40.389,-31.710,87.161,173.2885,0.7549,-16688.1360
C01180=37.311,-32.743,86.112,167.0986,-9.1514,-16691.2692
C01181=35.843,-34.176,86.067,168.4446,-12.1385,-16693.6362
C01182=35.014,-35.014,86.097,168.1689,-11.8314,-16695.0000
C01183=34.176,-35.842,86.067,167.8614,-11.5553,-16696.3630
C01184=32.743,-37.311,86.112,170.8503,-12.9018,-16698.7308
C01185=31.710,-40.389,87.161,-179.2449,-6.7109,-16701.8640
C01186=34.096,-44.548,89.719,179.2805,0.9468,-16702.5704
C01187=38.603,-50.345,93.033,179.4917,0.6633,-16702.5201
C01188=8.302,-62.896,93.033,-179.8904,-0.8284,-16732.4807
C01189=7.391,-55.610,89.719,-179.8393,-1.1782,-16732.4293
C01190=6.137,-50.981,87.161,175.7739,5.2863,-16733.1359
C01191=3.230,-49.536,86.112,164.5770,2.7513,-16736.2693
C01192=1.179,-49.510,86.067,163.4764,-0.4305,-16738.6359
C01193=0.000,-49.517,86.097,163.4981,-0.0002,-16740.0000
C01194=0.000,-49.517,86.097,163.4981,-0.0002,-16740.0000
C01195=-1.178,-49.510,86.067,163.4764,0.4306,-16741.3630
C01196=-3.231,-49.536,86.112,164.5779,-2.7529,-16743.7318
C01197=-6.137,-50.981,87.161,175.7745,-5.2860,-16746.8641
C01198=-7.391,-55.610,89.719,-179.8393,1.1782,-16747.5707
C01199=-8.302,-62.896,93.033,-179.8904,0.8284,-16747.5193
C01200=-38.603,-50.345,93.033,179.4917,-0.6633,-16777.4799
C01201=-34.096,-44.548,89.719,179.2805,-0.9468,-16777.4296
C01202=-31.710,-40.389,87.161,-179.2451,6.7115,-16778.1360
C01203=-32.743,-37.311,86.112,170.8486,12.9014,-16781.2692
C01204=-34.176,-35.843,86.067,167.8615,11.5554,-16783.6362
C01205=-35.014,-35.014,86.097,168.1686,11.8311,-16785.0000
C01206=-35.842,-34.176,86.067,168.4447,12.1386,-16786.3630
C01207=-37.311,-32.743,86.112,167.0982,9.1497,-16788.7308
C01208=-40.389,-31.710,87.161,173.2891,-0.7551,-16791.8640
C01209=-44.548,-34.096,89.719,-179.0532,0.7195,-16792.5704
C01210=-50.345,-38.603,93.033,-179.3367,0.5083,-16792.5201
C01211=-62.896,-8.302,93.033,179.1716,-0.1096,-16822.4807
C01212=-55.610,-7.391,89.719,178.8218,-0.1607,-16822.4293
C01213=-50.981,-6.137,87.161,-174.7137,4.2261,-16823.1359
C01214=-49.536,-3.230,86.112,-177.2487,15.4230,-16826.2693
C01215=-49.510,-1.179,86.067,179.5695,16.5236,-16828.6359
C01216=-49.517,0.000,86.097,179.9998,16.5019,-16830.0000
C01217=-49.510,1.178,86.067,-179.5694,16.5236,-16831.3630
C01218=-49.536,3.231,86.112,177.2471,15.4221,-16833.7318
C01219=-50.981,6.137,87.161,174.7140,4.2255,-16836.8641
C01220=-55.610,7.391,89.719,-178.8218,-0.1607,-16837.5707
C01221=-62.896,8.302,93.033,-179.1716,-0.1096,-16837.5193
C01222=-50.345,38.603,93.033,179.3367,0.5083,-16867.4799
C01223=-44.548,34.096,89.719,179.0532,0.7195,-16867.4296
C01224=-40.389,31.710,87.161,-173.2885,-0.7549,-16868.1360
C01225=-37.311,32.743,86.112,-167.0986,9.1514,-16871.2692
C01226=-35.843,34.176,86.067,-168.4446,12.1385,-16873.6362
C01227=-35.014,35.014,86.097,-168.1689,11.8314,-16875.0000
C01228=-34.176,35.842,86.067,-167.8614,11.5553,-16876.3630
C01229=-32.743,37.311,86.112,-170.8503,12.9018,-16878.7308
C01230=-31.710,40.389,87.161,179.2449,6.7109,-16881.8640
C01231=-34.096,44.548,89.719,-179.2805,-0.9468,-16882.5704
C01232=-38.603,50.345,93.033,-179.4917,-0.6633,-16882.5201
C01233=-8.302,62.896,93.033,179.8904,0.8284,-16912.4807
C01234=-7.391,55.610,89.719,179.8393,1.1782,-16912.4293
C01235=-6.137,50.981,87.161,-175.7745,-5.2860,-16913.1359
C01236=-3.231,49.536,86.112,-164.5779,-2.7529,-16916.2682
C01237=-1.178,49.510,86.067,-163.4764,0.4306,-16918.6370
C01238=0.000,49.517,86.097,-163.4981,-0.0002,-16920.0000
C01239=0.000,48.949,88.223,-166.6221,-0.0001,-16920.0000
C01240=1.127,48.942,88.191,-166.5931,-0.3233,-16921.3191
C01241=3.143,48.975,88.238,-167.5529,2.2752,-16923.6720
C01242=6.042,50.501,89.306,-176.8083,4.0597,-16926.8225
C01243=7.312,55.314,91.898,179.8925,-0.8037,-16927.5303
C01244=8.270,62.805,95.231,179.9710,-0.2201,-16927.5014
C01245=38.562,50.258,95.231,-179.8648,0.1762,-16957.4983
C01246=33.942,44.284,91.898,-179.5076,0.6443,-16957.4688
C01247=31.437,39.982,89.306,179.3837,-5.1210,-16958.1772
C01248=32.408,36.853,88.238,-172.7068,-10.4353,-16961.3279
C01249=33.811,35.404,88.191,-170.2108,-9.3446,-16963.6816
C01250=34.612,34.612,88.223,-170.4539,-9.5459,-16965.0000
C01251=35.404,33.811,88.191,-170.6554,-9.7892,-16966.3184
C01252=36.854,32.408,88.238,-169.5644,-7.2918,-16968.6728
C01253=39.982,31.437,89.306,-174.8795,0.6164,-16971.8228
C01254=44.284,33.942,91.898,179.3557,-0.4924,-16972.5312
C01255=50.258,38.562,95.231,179.8238,-0.1352,-16972.5017
C01256=62.805,8.270,95.231,-179.7799,0.0290,-17002.4986
C01257=55.314,7.312,91.898,-179.1963,0.1075,-17002.4697
C01258=50.501,6.042,89.306,175.9403,-3.1917,-17003.1775
C01259=48.975,3.143,88.238,177.7248,-12.4471,-17006.3280
C01260=48.942,1.127,88.191,-179.6767,-13.4069,-17008.6809
C01261=48.949,0.000,88.223,-179.9999,-13.3779,-17010.0000
C01262=48.942,-1.126,88.191,179.6767,-13.4069,-17011.3180
C01263=48.976,-3.143,88.238,-177.7235,-12.4463,-17013.6719
C01264=50.501,-6.042,89.306,-175.9405,-3.1912,-17016.8225
C01265=55.314,-7.312,91.898,179.1963,0.1075,-17017.5303
C01266=62.805,-8.270,95.231,179.7799,0.0290,-17017.5014
C01267=50.258,-38.562,95.231,-179.8238,-0.1352,-17047.4983
C01268=44.284,-33.942,91.898,-179.3557,-0.4924,-17047.4688
C01269=39.982,-31.437,89.306,174.8790,0.6163,-17048.1772
C01270=36.853,-32.408,88.238,169.5647,-7.2932,-17051.3279
C01271=35.404,-33.811,88.191,170.6554,-9.7892,-17053.6816
C01272=34.612,-34.612,88.223,170.4541,-9.5461,-17055.0000
C01273=33.811,-35.404,88.191,170.2108,-9.3446,-17056.3184
C01274=32.408,-36.854,88.238,172.7082,-10.4356,-17058.6728
C01275=31.437,-39.982,89.306,-179.3836,-5.1205,-17061.8228
C01276=33.942,-44.284,91.898,179.5076,0.6443,-17062.5312
C01277=38.562,-50.258,95.231,179.8648,0.1762,-17062.5017
C01278=8.270,-62.805,95.231,-179.9710,-0.2201,-17092.4986
C01279=7.312,-55.314,91.898,-179.8925,-0.8037,-17092.4697
C01280=6.042,-50.501,89.306,176.8083,4.0597,-17093.1775
C01281=3.143,-48.975,88.238,167.5529,2.2752,-17096.3280
C01282=1.127,-48.942,88.191,166.5931,-0.3233,-17098.6809
C01283=0.000,-48.949,88.223,166.6221,-0.0001,-17100.0000
C01284=0.000,-48.949,88.223,166.6221,-0.0001,-17100.0000
C01285=-1.126,-48.942,88.191,166.5931,0.3233,-17101.3180
C01286=-3.143,-48.976,88.238,167.5537,-2.2765,-17103.6719
C01287=-6.042,-50.501,89.306,176.8088,-4.0595,-17106.8225
C01288=-7.312,-55.314,91.898,-179.8925,0.8037,-17107.5303
C01289=-8.270,-62.805,95.231,-179.9710,0.2201,-17107.5014
C01290=-38.562,-50.258,95.231,179.8648,-0.1762,-17137.4983
C01291=-33.942,-44.284,91.898,179.5076,-0.6443,-17137.4688
C01292=-31.437,-39.982,89.306,-179.3837,5.1210,-17138.1772
C01293=-32.408,-36.853,88.238,172.7068,10.4353,-17141.3279
C01294=-33.811,-35.404,88.191,170.2108,9.3446,-17143.6816
C01295=-34.612,-34.612,88.223,170.4539,9.5459,-17145.0000
C01296=-35.404,-33.811,88.191,170.6554,9.7892,-17146.3184
C01297=-36.854,-32.408,88.238,169.5644,7.2918,-17148.6728
C01298=-39.982,-31.437,89.306,174.8795,-0.6164,-17151.8228
C01299=-44.284,-33.942,91.898,-179.3557,0.4924,-17152.5312
C01300=-50.258,-38.562,95.231,-179.8238,0.1352,-17152.5017
C01301=-62.805,-8.270,95.231,179.7799,-0.0290,-17182.4986
C01302=-55.314,-7.312,91.898,179.1963,-0.1075,-17182.4697
C01303=-50.501,-6.042,89.306,-175.9403,3.1917,-17183.1775
C01304=-48.975,-3.143,88.238,-177.7248,12.4471,-17186.3280
C01305=-48.942,-1.127,88.191,179.6767,13.4069,-17188.6809
C01306=-48.949,0.000,88.223,179.9999,13.3779,-17190.0000
C01307=-48.942,1.126,88.191,-179.6767,13.4069,-17191.3180
C01308=-48.976,3.143,88.238,177.7235,12.4463,-17193.6719
C01309=-50.501,6.042,89.306,175.9405,3.1912,-17196.8225
C01310=-55.314,7.312,91.898,-179.1963,-0.1075,-17197.5303
C01311=-62.805,8.270,95.231,-179.7799,-0.0290,-17197.5014
C01312=-50.258,38.562,95.231,179.8238,0.1352,-17227.4983
C01313=-44.284,33.942,91.898,179.3557,0.4924,-17227.4688
C01314=-39.982,31.437,89.306,-174.8790,-0.6163,-17228.1772
C01315=-36.853,32.408,88.238,-169.5647,7.2932,-17231.3279
C01316=-35.404,33.811,88.191,-170.6554,9.7892,-17233.6816
C01317=-34.612,34.612,88.223,-170.4541,9.5461,-17235.0000
C01318=-33.811,35.404,88.191,-170.2108,9.3446,-17236.3184
C01319=-32.408,36.854,88.238,-172.7082,10.4356,-17238.6728
C01320=-31.437,39.982,89.306,179.3836,5.1205,-17241.8228
C01321=-33.942,44.284,91.898,-179.5076,-0.6443,-17242.5312
C01322=-38.562,50.258,95.231,-179.8648,-0.1762,-17242.5017
C01323=-8.270,62.805,95.231,179.9710,0.2201,-17272.4986
C01324=-7.312,55.314,91.898,179.8925,0.8037,-17272.4697
C01325=-6.042,50.501,89.306,-176.8088,-4.0595,-17273.1775
C01326=-3.143,48.976,88.238,-167.5537,-2.2765,-17276.3281
C01327=-1.126,48.942,88.191,-166.5931,0.3233,-17278.6820
C01328=0.000,48.949,88.223,-166.6221,-0.0001,-17280.0000
C01329=0.000,48.503,90.377,-170.0356,-0.0001,-17280.0000
C01330=1.086,48.496,90.345,-169.9984,-0.2252,-17281.2828
C01331=3.075,48.536,90.393,-170.7679,1.7188,-17283.6251
C01332=5.972,50.143,91.476,-177.8365,2.7864,-17286.7919
C01333=7.266,55.138,94.090,179.9489,-0.3871,-17287.5071
C01334=33.851,44.126,94.090,-179.7624,0.3099,-17317.4934
C01335=31.234,39.679,91.476,179.5587,-3.4981,-17318.2087
C01336=32.146,36.494,90.393,-174.6463,-7.7532,-17321.3754
C01337=33.524,35.059,90.345,-172.7350,-6.9514,-17323.7178
C01338=34.297,34.297,90.377,-172.9184,-7.0815,-17325.0000
C01339=35.059,33.525,90.345,-173.0486,-7.2649,-17326.2813
C01340=36.495,32.146,90.393,-172.2466,-5.3526,-17328.6253
C01341=39.679,31.234,91.476,-176.5023,0.4414,-17331.7913
C01342=44.126,33.851,94.090,179.6901,-0.2376,-17332.5066
C01343=55.138,7.266,94.090,-179.6129,0.0511,-17362.4929
C01344=50.143,5.972,91.476,177.2136,-2.1635,-17363.2081
C01345=48.536,3.075,90.393,178.2812,-9.2321,-17366.3749
C01346=48.496,1.086,90.345,-179.7748,-10.0016,-17368.7172
C01347=48.503,0.000,90.377,-179.9999,-9.9644,-17370.0000
C01348=48.496,-1.085,90.345,179.7749,-10.0016,-17371.2817
C01349=48.536,-3.075,90.393,-178.2802,-9.2314,-17373.6251
C01350=50.143,-5.972,91.476,-177.2137,-2.1632,-17376.7919
C01351=55.138,-7.266,94.090,179.6129,0.0511,-17377.5071
C01352=44.126,-33.851,94.090,-179.6901,-0.2376,-17407.4934
C01353=39.679,-31.234,91.476,176.5019,0.4413,-17408.2087
C01354=36.494,-32.146,90.393,172.2468,-5.3537,-17411.3754
C01355=35.059,-33.524,90.345,173.0486,-7.2650,-17413.7178
C01356=34.297,-34.297,90.377,172.9185,-7.0816,-17415.0000
C01357=33.525,-35.059,90.345,172.7351,-6.9514,-17416.2813
C01358=32.146,-36.495,90.393,174.6474,-7.7534,-17418.6253
C01359=31.234,-39.679,91.476,-179.5586,-3.4977,-17421.7913
C01360=33.851,-44.126,94.090,179.7624,0.3099,-17422.5066
C01361=7.266,-55.138,94.090,-179.9489,-0.3871,-17452.4929
C01362=5.972,-50.143,91.476,177.8365,2.7864,-17453.2081
C01363=3.075,-48.536,90.393,170.7679,1.7188,-17456.3749
C01364=1.086,-48.496,90.345,169.9984,-0.2252,-17458.7172
C01365=0.000,-48.503,90.377,170.0356,-0.0001,-17460.0000
C01366=0.000,-48.503,90.377,170.0356,-0.0001,-17460.0000
C01367=-1.085,-48.496,90.345,169.9984,0.2251,-17461.2817
C01368=-3.075,-48.536,90.393,170.7686,-1.7198,-17463.6251
C01369=-5.972,-50.143,91.476,177.8368,-2.7863,-17466.7919
C01370=-7.266,-55.138,94.090,-179.9489,0.3871,-17467.5071
C01371=-33.851,-44.126,94.090,179.7624,-0.3099,-17497.4934
C01372=-31.234,-39.679,91.476,-179.5587,3.4981,-17498.2087
C01373=-32.146,-36.494,90.393,174.6463,7.7532,-17501.3754
C01374=-33.524,-35.059,90.345,172.7350,6.9514,-17503.7178
C01375=-34.297,-34.297,90.377,172.9184,7.0815,-17505.0000
C01376=-35.059,-33.525,90.345,173.0486,7.2649,-17506.2813
C01377=-36.495,-32.146,90.393,172.2466,5.3526,-17508.6253
C01378=-39.679,-31.234,91.476,176.5023,-0.4414,-17511.7913
C01379=-44.126,-33.851,94.090,-179.6901,0.2376,-17512.5066
C01380=-55.138,-7.266,94.090,179.6129,-0.0511,-17542.4929
C01381=-50.143,-5.972,91.476,-177.2136,2.1635,-17543.2081
C01382=-48.536,-3.075,90.393,-178.2812,9.2321,-17546.3749
C01383=-48.496,-1.086,90.345,179.7748,10.0016,-17548.7172
C01384=-48.503,0.000,90.377,179.9999,9.9644,-17550.0000
C01385=-48.496,1.085,90.345,-179.7749,10.0016,-17551.2817
C01386=-48.536,3.075,90.393,178.2802,9.2314,-17553.6251
C01387=-50.143,5.972,91.476,177.2137,2.1632,-17556.7919
C01388=-55.138,7.266,94.090,-179.6129,-0.0511,-17557.5071
C01389=-44.126,33.851,94.090,179.6901,0.2376,-17587.4934
C01390=-39.679,31.234,91.476,-176.5019,-0.4413,-17588.2087
C01391=-36.494,32.146,90.393,-172.2468,5.3537,-17591.3754
C01392=-35.059,33.524,90.345,-173.0486,7.2650,-17593.7178
C01393=-34.297,34.297,90.377,-172.9185,7.0816,-17595.0000
C01394=-33.525,35.059,90.345,-172.7351,6.9514,-17596.2813
C01395=-32.146,36.495,90.393,-174.6474,7.7534,-17598.6253
C01396=-31.234,39.679,91.476,179.5586,3.4977,-17601.7913
C01397=-33.851,44.126,94.090,-179.7624,-0.3099,-17602.5066
C01398=-7.266,55.138,94.090,179.9489,0.3871,-17632.4929
C01399=-5.972,50.143,91.476,-177.8368,-2.7863,-17633.2081
C01400=-3.075,48.536,90.393,-170.7686,-1.7198,-17636.3749
C01401=-1.085,48.496,90.345,-169.9984,0.2251,-17638.7183
C01402=0.000,48.503,90.377,-170.0356,-0.0001,-17640.0000
C01403=0.000,48.191,92.555,-173.7266,-0.0000,-17640.0000
C01404=1.057,48.183,92.523,-173.6804,-0.1349,-17641.2567
C01405=3.027,48.229,92.571,-174.2129,1.0909,-17643.5913
C01406=5.927,49.917,93.664,-178.8724,1.4637,-17646.7714
C01407=31.106,39.488,93.664,179.7623,-1.8320,-17678.2287
C01408=31.963,36.244,92.571,-176.6691,-4.8658,-17681.4086
C01409=33.323,34.818,92.523,-175.4275,-4.3829,-17683.7431
C01410=34.076,34.076,92.555,-175.5552,-4.4448,-17685.0000
C01411=34.818,33.324,92.523,-175.6171,-4.5724,-17686.2560
C01412=36.244,31.963,92.571,-175.1341,-3.3301,-17688.5914
C01413=39.488,31.106,93.664,-178.1682,0.2378,-17691.7713
C01414=49.917,5.927,93.664,178.5363,-1.1276,-17723.2286
C01415=48.229,3.027,92.571,178.9091,-5.7871,-17726.4087
C01416=48.183,1.057,92.523,-179.8651,-6.3196,-17728.7433
C01417=48.191,0.000,92.555,-180.0000,-6.2734,-17730.0000
C01418=48.183,-1.057,92.523,179.8652,-6.3196,-17731.2567
C01419=48.229,-3.027,92.571,-178.9086,-5.7866,-17733.5913
C01420=49.918,-5.927,93.664,-178.5365,-1.1274,-17736.7713
C01421=39.488,-31.106,93.664,178.1680,0.2377,-17768.2287
C01422=36.244,-31.963,92.571,175.1342,-3.3309,-17771.4086
C01423=34.818,-33.323,92.523,175.6171,-4.5725,-17773.7431
C01424=34.076,-34.076,92.555,175.5552,-4.4448,-17775.0000
C01425=33.324,-34.818,92.523,175.4276,-4.3829,-17776.2560
C01426=31.963,-36.244,92.571,176.6699,-4.8659,-17778.5914
C01427=31.106,-39.488,93.664,-179.7622,-1.8318,-17781.7713
C01428=5.927,-49.917,93.664,178.8724,1.4637,-17813.2286
C01429=3.027,-48.229,92.571,174.2129,1.0909,-17816.4087
C01430=1.057,-48.183,92.523,173.6804,-0.1349,-17818.7433
C01431=0.000,-48.191,92.555,173.7266,-0.0000,-17820.0000
C01432=0.000,-48.191,92.555,173.7266,-0.0000,-17820.0000
C01433=-1.057,-48.183,92.523,173.6804,0.1348,-17821.2567
C01434=-3.027,-48.229,92.571,174.2134,-1.0914,-17823.5913
C01435=-5.927,-49.918,93.664,178.8726,-1.4635,-17826.7713
C01436=-31.106,-39.488,93.664,-179.7623,1.8320,-17858.2287
C01437=-31.963,-36.244,92.571,176.6691,4.8658,-17861.4086
C01438=-33.323,-34.818,92.523,175.4275,4.3829,-17863.7431
C01439=-34.076,-34.076,92.555,175.5552,4.4448,-17865.0000
C01440=-34.818,-33.324,92.523,175.6171,4.5724,-17866.2560
C01441=-36.244,-31.963,92.571,175.1341,3.3301,-17868.5914
C01442=-39.488,-31.106,93.664,178.1682,-0.2378,-17871.7713
C01443=-49.917,-5.927,93.664,-178.5363,1.1276,-17903.2286
C01444=-48.229,-3.027,92.571,-178.9091,5.7871,-17906.4087
C01445=-48.183,-1.057,92.523,179.8651,6.3196,-17908.7433
C01446=-48.191,0.000,92.555,180.0000,6.2734,-17910.0000
C01447=-48.183,1.057,92.523,-179.8652,6.3196,-17911.2567
C01448=-48.229,3.027,92.571,178.9086,5.7866,-17913.5913
C01449=-49.918,5.927,93.664,178.5365,1.1274,-17916.7713
C01450=-39.488,31.106,93.664,-178.1680,-0.2377,-17948.2287
C01451=-36.244,31.963,92.571,-175.1342,3.3309,-17951.4086
C01452=-34.818,33.323,92.523,-175.6171,4.5725,-17953.7431
C01453=-34.076,34.076,92.555,-175.5552,4.4448,-17955.0000
C01454=-33.324,34.818,92.523,-175.4276,4.3829,-17956.2560
C01455=-31.963,36.244,92.571,-176.6699,4.8659,-17958.5914
C01456=-31.106,39.488,93.664,179.7622,1.8318,-17961.7713
C01457=-5.927,49.918,93.664,-178.8726,-1.4635,-17993.2287
C01458=-3.027,48.229,92.571,-174.2134,-1.0914,-17996.4087
C01459=-1.057,48.183,92.523,-173.6804,0.1348,-17998.7433
C01460=0.000,48.191,92.555,-173.7266,-0.0000,-18000.0000
C01461=0.000,48.026,94.749,-177.6660,-0.0000,-18000.0000
C01462=1.042,48.016,94.716,-177.6104,-0.0495,-18001.2432
C01463=3.002,48.067,94.764,-177.8674,0.4046,-18003.5737
C01464=5.911,49.834,95.862,-179.9324,0.0880,-18006.7645
C01465=31.058,39.418,95.862,179.9856,-0.1101,-18038.2351
C01466=31.866,36.111,94.764,-178.7776,-1.7942,-18041.4267
C01467=33.216,34.689,94.716,-178.2749,-1.6552,-18043.7573
C01468=33.959,33.959,94.749,-178.3492,-1.6508,-18045.0000
C01469=34.689,33.216,94.716,-178.3447,-1.7251,-18046.2427
C01470=36.111,31.865,94.764,-178.2059,-1.2221,-18048.5742
C01471=39.418,31.058,95.862,-179.8900,0.0144,-18051.7649
C01472=49.834,5.911,95.862,179.9120,-0.0676,-18083.2355
C01473=48.067,3.002,94.764,179.5954,-2.1326,-18086.4263
C01474=48.016,1.042,94.716,-179.9505,-2.3896,-18088.7568
C01475=48.026,0.000,94.749,-180.0000,-2.3340,-18090.0000
C01476=48.016,-1.041,94.716,179.9506,-2.3896,-18091.2420
C01477=48.067,-3.002,94.764,-179.5952,-2.1323,-18093.5737
C01478=49.834,-5.911,95.862,-179.9120,-0.0676,-18096.7645
C01479=39.418,-31.058,95.862,179.8899,0.0144,-18128.2351
C01480=36.111,-31.866,94.764,178.2058,-1.2224,-18131.4267
C01481=34.689,-33.216,94.716,178.3448,-1.7251,-18133.7573
C01482=33.959,-33.959,94.749,178.3492,-1.6508,-18135.0000
C01483=33.216,-34.689,94.716,178.2749,-1.6553,-18136.2427
C01484=31.865,-36.111,94.764,178.7779,-1.7941,-18138.5742
C01485=31.058,-39.418,95.862,-179.9856,-0.1100,-18141.7649
C01486=5.911,-49.834,95.862,179.9324,0.0880,-18173.2355
C01487=3.002,-48.067,94.764,177.8674,0.4046,-18176.4263
C01488=1.042,-48.016,94.716,177.6104,-0.0495,-18178.7568
C01489=0.000,-48.026,94.749,177.6660,-0.0000,-18180.0000
C01490=0.000,-48.026,94.749,177.6660,-0.0000,-18180.0000
C01491=-1.041,-48.016,94.716,177.6104,0.0494,-18181.2420
C01492=-3.002,-48.067,94.764,177.8677,-0.4048,-18183.5737
C01493=-5.911,-49.834,95.862,179.9324,-0.0880,-18186.7645
C01494=-31.058,-39.418,95.862,-179.9856,0.1101,-18218.2351
C01495=-31.866,-36.111,94.764,178.7776,1.7942,-18221.4267
C01496=-33.216,-34.689,94.716,178.2749,1.6552,-18223.7573
C01497=-33.959,-33.959,94.749,178.3492,1.6508,-18225.0000
C01498=-34.689,-33.216,94.716,178.3447,1.7251,-18226.2427
C01499=-36.111,-31.865,94.764,178.2059,1.2221,-18228.5742
C01500=-39.418,-31.058,95.862,179.8900,-0.0144,-18231.7649
C01501=-49.834,-5.911,95.862,-179.9120,0.0676,-18263.2355
C01502=-48.067,-3.002,94.764,-179.5954,2.1326,-18266.4263
C01503=-48.016,-1.042,94.716,179.9505,2.3896,-18268.7568
C01504=-48.026,0.000,94.749,180.0000,2.3340,-18270.0000
C01505=-48.016,1.041,94.716,-179.9506,2.3896,-18271.2420
C01506=-48.067,3.002,94.764,179.5952,2.1323,-18273.5737
C01507=-49.834,5.911,95.862,179.9120,0.0676,-18276.7645
C01508=-39.418,31.058,95.862,-179.8899,-0.0144,-18308.2351
C01509=-36.111,31.866,94.764,-178.2058,1.2224,-18311.4267
C01510=-34.689,33.216,94.716,-178.3448,1.7251,-18313.7573
C01511=-33.959,33.959,94.749,-178.3492,1.6508,-18315.0000
C01512=-33.216,34.689,94.716,-178.2749,1.6553,-18316.2427
C01513=-31.865,36.111,94.764,-178.7779,1.7941,-18318.5742
C01514=-31.058,39.418,95.862,179.9856,0.1100,-18321.7649
C01515=-5.911,49.834,95.862,-179.9324,-0.0880,-18353.2355
C01516=-3.002,48.067,94.764,-177.8677,-0.4048,-18356.4263
C01517=-1.041,48.016,94.716,-177.6104,0.0494,-18358.7580
C01518=0.000,48.026,94.749,-177.6660,-0.0000,-18360.0000
///TOOL 0
///POSTYPE ANGLE
///ANGLE
EC00000=0.0000,14256.8795
EC00001=0.0000,14256.8537
EC00002=0.0000,14257.6887
EC00003=0.0000,14260.6829
EC00004=0.0000,14263.1899
EC00005=0.0000,14265.0000
EC00006=0.0000,14266.8101
EC00007=0.0000,14269.3178
EC00008=0.0000,14272.3119
EC00009=0.0000,14273.1463
EC00010=0.0000,14273.1205
EC00011=0.0000,14272.9934
EC00012=0.0000,14272.8957
EC00013=0.0000,14272.9735
EC00014=0.0000,14274.6500
EC00015=0.0000,14277.6087
EC00016=0.0000,14281.3401
EC00017=0.0000,14285.4161
EC00018=0.0000,14289.5839
EC00019=0.0000,14293.6602
EC00020=0.0000,14297.3912
EC00021=0.0000,14300.3496
EC00022=0.0000,14302.0267
EC00023=0.0000,14302.1045
EC00024=0.0000,14302.0068
EC00025=0.0000,14301.8791
EC00026=0.0000,14301.8541
EC00027=0.0000,14302.6890
EC00028=0.0000,14305.6832
EC00029=0.0000,14308.1896
EC00030=0.0000,14310.0000
EC00031=0.0000,14311.8094
EC00032=0.0000,14314.3178
EC00033=0.0000,14317.3110
EC00034=0.0000,14318.1459
EC00035=0.0000,14318.1209
EC00036=0.0000,14317.9932
EC00037=0.0000,14317.8955
EC00038=0.0000,14317.9733
EC00039=0.0000,14319.6504
EC00040=0.0000,14322.6088
EC00041=0.0000,14326.3398
EC00042=0.0000,14330.4161
EC00043=0.0000,14334.5839
EC00044=0.0000,14338.6599
EC00045=0.0000,14342.3913
EC00046=0.0000,14345.3500
EC00047=0.0000,14347.0265
EC00048=0.0000,14347.1043
EC00049=0.0000,14347.0066
EC00050=0.0000,14346.8795
EC00051=0.0000,14346.8537
EC00052=0.0000,14347.6887
EC00053=0.0000,14350.6829
EC00054=0.0000,14353.1899
EC00055=0.0000,14355.0000
EC00056=0.0000,14356.8101
EC00057=0.0000,14359.3178
EC00058=0.0000,14362.3119
EC00059=0.0000,14363.1463
EC00060=0.0000,14363.1205
EC00061=0.0000,14362.9934
EC00062=0.0000,14362.8957
EC00063=0.0000,14362.9735
EC00064=0.0000,14364.6500
EC00065=0.0000,14367.6087
EC00066=0.0000,14371.3401
EC00067=0.0000,14375.4161
EC00068=0.0000,14379.5839
EC00069=0.0000,14383.6602
EC00070=0.0000,14387.3912
EC00071=0.0000,14390.3496
EC00072=0.0000,14392.0267
EC00073=0.0000,14392.1045
EC00074=0.0000,14392.0068
EC00075=0.0000,14391.8791
EC00076=0.0000,14391.8541
EC00077=0.0000,14392.6890
EC00078=0.0000,14395.6822
EC00079=0.0000,14398.1906
EC00080=0.0000,14400.0000
EC00081=0.0000,14400.0000
EC00082=0.0000,14401.7406
EC00083=0.0000,14404.2255
EC00084=0.0000,14407.2387
EC00085=0.0000,14408.0440
EC00086=0.0000,14407.9981
EC00087=0.0000,14407.8709
EC00088=0.0000,14407.7793
EC00089=0.0000,14407.8555
EC00090=0.0000,14409.5452
EC00091=0.0000,14412.5282
EC00092=0.0000,14416.2898
EC00093=0.0000,14420.3994
EC00094=0.0000,14424.6009
EC00095=0.0000,14428.7101
EC00096=0.0000,14432.4718
EC00097=0.0000,14435.4547
EC00098=0.0000,14437.1446
EC00099=0.0000,14437.2208
EC00100=0.0000,14437.1290
EC00101=0.0000,14437.0022
EC00102=0.0000,14436.9563
EC00103=0.0000,14437.7605
EC00104=0.0000,14440.7744
EC00105=0.0000,14443.2595
EC00106=0.0000,14445.0000
EC00107=0.0000,14446.7398
EC00108=0.0000,14449.2256
EC00109=0.0000,14452.2395
EC00110=0.0000,14453.0437
EC00111=0.0000,14452.9978
EC00112=0.0000,14452.8710
EC00113=0.0000,14452.7792
EC00114=0.0000,14452.8554
EC00115=0.0000,14454.5453
EC00116=0.0000,14457.5282
EC00117=0.0000,14461.2899
EC00118=0.0000,14465.3991
EC00119=0.0000,14469.6006
EC00120=0.0000,14473.7102
EC00121=0.0000,14477.4718
EC00122=0.0000,14480.4548
EC00123=0.0000,14482.1445
EC00124=0.0000,14482.2207
EC00125=0.0000,14482.1291
EC00126=0.0000,14482.0019
EC00127=0.0000,14481.9560
EC00128=0.0000,14482.7613
EC00129=0.0000,14485.7745
EC00130=0.0000,14488.2594
EC00131=0.0000,14490.0000
EC00132=0.0000,14491.7396
EC00133=0.0000,14494.2255
EC00134=0.0000,14497.2387
EC00135=0.0000,14498.0440
EC00136=0.0000,14497.9981
EC00137=0.0000,14497.8709
EC00138=0.0000,14497.7793
EC00139=0.0000,14497.8555
EC00140=0.0000,14499.5452
EC00141=0.0000,14502.5282
EC00142=0.0000,14506.2898
EC00143=0.0000,14510.3994
EC00144=0.0000,14514.6009
EC00145=0.0000,14518.7101
EC00146=0.0000,14522.4718
EC00147=0.0000,14525.4547
EC00148=0.0000,14527.1446
EC00149=0.0000,14527.2208
EC00150=0.0000,14527.1290
EC00151=0.0000,14527.0022
EC00152=0.0000,14526.9563
EC00153=0.0000,14527.7605
EC00154=0.0000,14530.7744
EC00155=0.0000,14533.2595
EC00156=0.0000,14535.0000
EC00157=0.0000,14536.7398
EC00158=0.0000,14539.2256
EC00159=0.0000,14542.2395
EC00160=0.0000,14543.0437
EC00161=0.0000,14542.9978
EC00162=0.0000,14542.8710
EC00163=0.0000,14542.7792
EC00164=0.0000,14542.8554
EC00165=0.0000,14544.5453
EC00166=0.0000,14547.5282
EC00167=0.0000,14551.2899
EC00168=0.0000,14555.3991
EC00169=0.0000,14559.6006
EC00170=0.0000,14563.7102
EC00171=0.0000,14567.4718
EC00172=0.0000,14570.4548
EC00173=0.0000,14572.1445
EC00174=0.0000,14572.2207
EC00175=0.0000,14572.1291
EC00176=0.0000,14572.0019
EC00177=0.0000,14571.9560
EC00178=0.0000,14572.7613
EC00179=0.0000,14575.7745
EC00180=0.0000,14578.2594
EC00181=0.0000,14580.0000
EC00182=0.0000,14580.0000
EC00183=0.0000,14581.7396
EC00184=0.0000,14584.2255
EC00185=0.0000,14587.2387
EC00186=0.0000,14588.0440
EC00187=0.0000,14587.9981
EC00188=0.0000,14587.8709
EC00189=0.0000,14587.7793
EC00190=0.0000,14587.8555
EC00191=0.0000,14589.5452
EC00192=0.0000,14592.5282
EC00193=0.0000,14596.2898
EC00194=0.0000,14600.3994
EC00195=0.0000,14604.6009
EC00196=0.0000,14608.7101
EC00197=0.0000,14612.4718
EC00198=0.0000,14615.4547
EC00199=0.0000,14617.1446
EC00200=0.0000,14617.2208
EC00201=0.0000,14617.1290
EC00202=0.0000,14617.0022
EC00203=0.0000,14616.9563
EC00204=0.0000,14617.7605
EC00205=0.0000,14620.7744
EC00206=0.0000,14623.2595
EC00207=0.0000,14625.0000
EC00208=0.0000,14626.7398
EC00209=0.0000,14629.2256
EC00210=0.0000,14632.2395
EC00211=0.0000,14633.0437
EC00212=0.0000,14632.9978
EC00213=0.0000,14632.8710
EC00214=0.0000,14632.7792
EC00215=0.0000,14632.8554
EC00216=0.0000,14634.5453
EC00217=0.0000,14637.5282
EC00218=0.0000,14641.2899
EC00219=0.0000,14645.3991
EC00220=0.0000,14649.6006
EC00221=0.0000,14653.7102
EC00222=0.0000,14657.4718
EC00223=0.0000,14660.4548
EC00224=0.0000,14662.1445
EC00225=0.0000,14662.2207
EC00226=0.0000,14662.1291
EC00227=0.0000,14662.0019
EC00228=0.0000,14661.9560
EC00229=0.0000,14662.7613
EC00230=0.0000,14665.7745
EC00231=0.0000,14668.2594
EC00232=0.0000,14670.0000
EC00233=0.0000,14671.7396
EC00234=0.0000,14674.2255
EC00235=0.0000,14677.2387
EC00236=0.0000,14678.0440
EC00237=0.0000,14677.9981
EC00238=0.0000,14677.8709
EC00239=0.0000,14677.7793
EC00240=0.0000,14677.8555
EC00241=0.0000,14679.5452
EC00242=0.0000,14682.5282
EC00243=0.0000,14686.2898
EC00244=0.0000,14690.3994
EC00245=0.0000,14694.6009
EC00246=0.0000,14698.7101
EC00247=0.0000,14702.4718
EC00248=0.0000,14705.4547
EC00249=0.0000,14707.1446
EC00250=0.0000,14707.2208
EC00251=0.0000,14707.1290
EC00252=0.0000,14707.0022
EC00253=0.0000,14706.9563
EC00254=0.0000,14707.7605
EC00255=0.0000,14710.7744
EC00256=0.0000,14713.2595
EC00257=0.0000,14715.0000
EC00258=0.0000,14716.7398
EC00259=0.0000,14719.2256
EC00260=0.0000,14722.2395
EC00261=0.0000,14723.0437
EC00262=0.0000,14722.9978
EC00263=0.0000,14722.8710
EC00264=0.0000,14722.7792
EC00265=0.0000,14722.8554
EC00266=0.0000,14724.5453
EC00267=0.0000,14727.5282
EC00268=0.0000,14731.2899
EC00269=0.0000,14735.3991
EC00270=0.0000,14739.6006
EC00271=0.0000,14743.7102
EC00272=0.0000,14747.4718
EC00273=0.0000,14750.4548
EC00274=0.0000,14752.1445
EC00275=0.0000,14752.2207
EC00276=0.0000,14752.1291
EC00277=0.0000,14752.0019
EC00278=0.0000,14751.9560
EC00279=0.0000,14752.7613
EC00280=0.0000,14755.7745
EC00281=0.0000,14758.2604
EC00282=0.0000,14760.0000
EC00283=0.0000,14760.0000
EC00284=0.0000,14761.6706
EC00285=0.0000,14764.1339
EC00286=0.0000,14767.1680
EC00287=0.0000,14767.9465
EC00288=0.0000,14767.8844
EC00289=0.0000,14767.7630
EC00290=0.0000,14767.6803
EC00291=0.0000,14767.7585
EC00292=0.0000,14769.4604
EC00293=0.0000,14772.4636
EC00294=0.0000,14776.2505
EC00295=0.0000,14780.3860
EC00296=0.0000,14784.6140
EC00297=0.0000,14788.7498
EC00298=0.0000,14792.5363
EC00299=0.0000,14795.5394
EC00300=0.0000,14797.2413
EC00301=0.0000,14797.3191
EC00302=0.0000,14797.2369
EC00303=0.0000,14797.1159
EC00304=0.0000,14797.0536
EC00305=0.0000,14797.8325
EC00306=0.0000,14800.8660
EC00307=0.0000,14803.3290
EC00308=0.0000,14805.0000
EC00309=0.0000,14806.6710
EC00310=0.0000,14809.1340
EC00311=0.0000,14812.1675
EC00312=0.0000,14812.9464
EC00313=0.0000,14812.8841
EC00314=0.0000,14812.7631
EC00315=0.0000,14812.6809
EC00316=0.0000,14812.7587
EC00317=0.0000,14814.4606
EC00318=0.0000,14817.4637
EC00319=0.0000,14821.2502
EC00320=0.0000,14825.3860
EC00321=0.0000,14829.6140
EC00322=0.0000,14833.7495
EC00323=0.0000,14837.5364
EC00324=0.0000,14840.5396
EC00325=0.0000,14842.2415
EC00326=0.0000,14842.3197
EC00327=0.0000,14842.2370
EC00328=0.0000,14842.1156
EC00329=0.0000,14842.0535
EC00330=0.0000,14842.8320
EC00331=0.0000,14845.8661
EC00332=0.0000,14848.3294
EC00333=0.0000,14850.0000
EC00334=0.0000,14851.6706
EC00335=0.0000,14854.1349
EC00336=0.0000,14857.1678
EC00337=0.0000,14857.9465
EC00338=0.0000,14857.8844
EC00339=0.0000,14857.7630
EC00340=0.0000,14857.6803
EC00341=0.0000,14857.7585
EC00342=0.0000,14859.4604
EC00343=0.0000,14862.4636
EC00344=0.0000,14866.2505
EC00345=0.0000,14870.3860
EC00346=0.0000,14874.6140
EC00347=0.0000,14878.7498
EC00348=0.0000,14882.5363
EC00349=0.0000,14885.5394
EC00350=0.0000,14887.2413
EC00351=0.0000,14887.3191
EC00352=0.0000,14887.2369
EC00353=0.0000,14887.1159
EC00354=0.0000,14887.0536
EC00355=0.0000,14887.8325
EC00356=0.0000,14890.8660
EC00357=0.0000,14893.3290
EC00358=0.0000,14895.0000
EC00359=0.0000,14896.6710
EC00360=0.0000,14899.1340
EC00361=0.0000,14902.1675
EC00362=0.0000,14902.9464
EC00363=0.0000,14902.8841
EC00364=0.0000,14902.7631
EC00365=0.0000,14902.6809
EC00366=0.0000,14902.7587
EC00367=0.0000,14904.4606
EC00368=0.0000,14907.4637
EC00369=0.0000,14911.2502
EC00370=0.0000,14915.3860
EC00371=0.0000,14919.6140
EC00372=0.0000,14923.7495
EC00373=0.0000,14927.5364
EC00374=0.0000,14930.5396
EC00375=0.0000,14932.2415
EC00376=0.0000,14932.3197
EC00377=0.0000,14932.2370
EC00378=0.0000,14932.1156
EC00379=0.0000,14932.0535
EC00380=0.0000,14932.8320
EC00381=0.0000,14935.8661
EC00382=0.0000,14938.3294
EC00383=0.0000,14940.0000
EC00384=0.0000,14940.0000
EC00385=0.0000,14941.6706
EC00386=0.0000,14944.1349
EC00387=0.0000,14947.1678
EC00388=0.0000,14947.9465
EC00389=0.0000,14947.8844
EC00390=0.0000,14947.7630
EC00391=0.0000,14947.6803
EC00392=0.0000,14947.7585
EC00393=0.0000,14949.4604
EC00394=0.0000,14952.4636
EC00395=0.0000,14956.2505
EC00396=0.0000,14960.3860
EC00397=0.0000,14964.6140
EC00398=0.0000,14968.7498
EC00399=0.0000,14972.5363
EC00400=0.0000,14975.5394
EC00401=0.0000,14977.2413
EC00402=0.0000,14977.3191
EC00403=0.0000,14977.2369
EC00404=0.0000,14977.1159
EC00405=0.0000,14977.0536
EC00406=0.0000,14977.8325
EC00407=0.0000,14980.8660
EC00408=0.0000,14983.3290
EC00409=0.0000,14985.0000
EC00410=0.0000,14986.6710
EC00411=0.0000,14989.1340
EC00412=0.0000,14992.1675
EC00413=0.0000,14992.9464
EC00414=0.0000,14992.8841
EC00415=0.0000,14992.7631
EC00416=0.0000,14992.6809
EC00417=0.0000,14992.7587
EC00418=0.0000,14994.4606
EC00419=0.0000,14997.4637
EC00420=0.0000,15001.2502
EC00421=0.0000,15005.3860
EC00422=0.0000,15009.6140
EC00423=0.0000,15013.7495
EC00424=0.0000,15017.5364
EC00425=0.0000,15020.5396
EC00426=0.0000,15022.2415
EC00427=0.0000,15022.3197
EC00428=0.0000,15022.2370
EC00429=0.0000,15022.1156
EC00430=0.0000,15022.0535
EC00431=0.0000,15022.8320
EC00432=0.0000,15025.8661
EC00433=0.0000,15028.3294
EC00434=0.0000,15030.0000
EC00435=0.0000,15031.6706
EC00436=0.0000,15034.1349
EC00437=0.0000,15037.1678
EC00438=0.0000,15037.9465
EC00439=0.0000,15037.8844
EC00440=0.0000,15037.7630
EC00441=0.0000,15037.6803
EC00442=0.0000,15037.7585
EC00443=0.0000,15039.4604
EC00444=0.0000,15042.4636
EC00445=0.0000,15046.2505
EC00446=0.0000,15050.3860
EC00447=0.0000,15054.6140
EC00448=0.0000,15058.7498
EC00449=0.0000,15062.5363
